// TwinCAT 3 PLC project Test_PLC
// ProgramVersion: 3.1.4026.20
// CompilerDefines: VISU_USEPROPERTYINFO
// libraries:
//   Tc2_Standard, * (Beckhoff Automation GmbH)
//   Tc2_System, * (Beckhoff Automation GmbH)
//   Tc3_Mc3PlanarMotion, * (Beckhoff Automation GmbH)
//   Tc3_Physics, * (Beckhoff Automation GmbH)
//   Tc3_XPlanarUtility, * (Beckhoff Automation GmbH)
//   VisuDialogs, * (System)
// project tree:
//   DUTs/ E_TrackName.TcDUT (not stored), ST_MoverFeedback.TcDUT, U_MoverFeedback.TcDUT
//   / GlobalTextList.TcGTLO, Nc_Task.TcTTO (not stored), PlcTask.TcTTO (not stored), Visualization Manager.TcVMO (not stored)
//   GVLs/ GVL.TcGVL
//   POUs/ FB_StateTrackMove.TcPOU, MAIN.TcPOU
//   VISUs/ TextList_TrackState.TcTLO, Visualization.TcVIS
// real-time tasks:
//   TASK PlcTask: cycle T#10ms, priority 20, ADS port 350
//   TASK Nc Task: cycle T#10ms, priority 1, ADS port 351
//   TASK XPlanar Task_5: cycle T#250us, priority 2, ADS port 352
//   TASK Job Task: cycle default, priority 3
//   TASK MC-Task (MET): cycle T#2ms, priority 4, ADS port 353
//   TASK MC-Task (MPT): cycle T#10ms, priority 5, ADS port 354
//   TASK Job Task_1: cycle default, priority 7
//   TASK MC-Task (MET)_1: cycle T#2ms, priority 8, ADS port 356
//   TASK MC-Task (MPT)_1: cycle T#10ms, priority 9, ADS port 357
//   TASK XPlanar Task_6: cycle T#250us, priority 6, ADS port 355
//   TASK XPlanar Task_7: cycle T#250us, priority 10, ADS port 358
//   TASK EIP Task: cycle T#10ms, priority 12, ADS port 301
// I/O:
//   DEVICE Device 4 (EtherCAT), AmsNetId 169.254.116.218.5.1
//     Term 1 (EK1100) [EK1100 EtherCAT Coupler (2A E-Bus)]
//       Term 2 (EL1008) [EL1008 8Ch. Dig. Input 24V, 3ms]
//       Term 3 (EL2008-0015) [EL2008-0015 8Ch. Dig. Output 24V DC, 0.35A, not short-circuit proof]
//       Term 4 (EL9576) [EL9576 Brake chopper terminal]
//       Term 5 (EL9227-6644) [EL9227-6644 Overcurrent protection 24V DC, 2Ch., 4A/4A, extended functionalities]
//       Term 6 (EL9227-6644) [EL9227-6644 Overcurrent protection 24V DC, 2Ch., 4A/4A, extended functionalities]
//       Term 7 (EL9011) [EL9011 End Terminal]
//   DEVICE Device 5 (EtherCAT), AmsNetId 169.254.116.218.6.1
//     Term 8 (APS4322-7000) [APS4322-7000 Drive]
//       Term 9 (APS4322-5000) [APS4322-5000 Feedback]
//     Term 10 (APS4322-7000) [APS4322-7000 Drive]
//       Term 11 (APS4322-5000) [APS4322-5000 Feedback]
//     Term 12 (APS4322-7000) [APS4322-7000 Drive]
//       Term 13 (APS4322-5000) [APS4322-5000 Feedback]
//     Term 14 (APS4322-7000) [APS4322-7000 Drive]
//       Term 15 (APS4322-5000) [APS4322-5000 Feedback]
//     Term 16 (APS4322-7000) [APS4322-7000 Drive]
//       Term 17 (APS4322-5000) [APS4322-5000 Feedback]
//     Term 18 (APS4322-7000) [APS4322-7000 Drive]
//       Term 19 (APS4322-5000) [APS4322-5000 Feedback]
//   DEVICE Device 6 (RT-Ethernet Adapter)
//   DEVICE Device 1 (TC3 EIP Adapter), AmsNetId 169.254.116.218.2.1
//     Box 20 (TC EtherNet/IP Slave)
// variable links:
//   Device 5 (EtherCAT) <-> TcCOM Objects/XPlanar/Part1/APS4322_P1_1
//     Term 14 (APS4322-7000)/APS Comm Inputs/CommStatusWord <-> Data Pointer/MoverCommStatusWord
//     Term 14 (APS4322-7000)/APS Comm Inputs/Data {1..4} <-> Data Pointer/MoverCommDataIn[{0..3}]  (4 links)
//     Term 14 (APS4322-7000)/APS Comm Outputs/CommControlWord <-> Data Pointer/MoverCommControlWord
//     Term 14 (APS4322-7000)/APS Comm Outputs/Data 1 <-> Data Pointer/MoverCommDataOut
//     Term 14 (APS4322-7000)/APS Diagdata/DC Link Voltage <-> Data Pointer/DcLinkVoltage
//     Term 14 (APS4322-7000)/APS Diagdata/Power supply current <-> Data Pointer/PowerSupplyCurrent
//     Term 14 (APS4322-7000)/APS Inputs/StatusWord <-> Data Pointer/PowerUnitStatusWord
//     Term 14 (APS4322-7000)/APS Outputs/ControlWord <-> Data Pointer/PowerUnitControlWord
//     Term 14 (APS4322-7000)/APS Outputs/Current D 0X0 <-> Data Pointer/DCurrentSetPoints[0]
//     Term 14 (APS4322-7000)/APS Outputs/Current D 0X1 <-> Data Pointer/DCurrentSetPoints[1]
//     Term 14 (APS4322-7000)/APS Outputs/Current D 0X2 <-> Data Pointer/DCurrentSetPoints[2]
//     Term 14 (APS4322-7000)/APS Outputs/Current D 1X0 <-> Data Pointer/DCurrentSetPoints[6]
//     Term 14 (APS4322-7000)/APS Outputs/Current D 1X1 <-> Data Pointer/DCurrentSetPoints[7]
//     Term 14 (APS4322-7000)/APS Outputs/Current D 1X2 <-> Data Pointer/DCurrentSetPoints[8]
//     Term 14 (APS4322-7000)/APS Outputs/Current D 2X0 <-> Data Pointer/DCurrentSetPoints[12]
//     Term 14 (APS4322-7000)/APS Outputs/Current D 2X1 <-> Data Pointer/DCurrentSetPoints[13]
//     Term 14 (APS4322-7000)/APS Outputs/Current D 2X2 <-> Data Pointer/DCurrentSetPoints[14]
//     Term 14 (APS4322-7000)/APS Outputs/Current D 3X0 <-> Data Pointer/DCurrentSetPoints[18]
//     Term 14 (APS4322-7000)/APS Outputs/Current D 3X1 <-> Data Pointer/DCurrentSetPoints[19]
//     Term 14 (APS4322-7000)/APS Outputs/Current D 3X2 <-> Data Pointer/DCurrentSetPoints[20]
//     Term 14 (APS4322-7000)/APS Outputs/Current D 0Y0 <-> Data Pointer/DCurrentSetPoints[3]
//     Term 14 (APS4322-7000)/APS Outputs/Current D 0Y1 <-> Data Pointer/DCurrentSetPoints[4]
//     Term 14 (APS4322-7000)/APS Outputs/Current D 0Y2 <-> Data Pointer/DCurrentSetPoints[5]
//     Term 14 (APS4322-7000)/APS Outputs/Current D 1Y0 <-> Data Pointer/DCurrentSetPoints[9]
//     Term 14 (APS4322-7000)/APS Outputs/Current D 1Y1 <-> Data Pointer/DCurrentSetPoints[10]
//     Term 14 (APS4322-7000)/APS Outputs/Current D 1Y2 <-> Data Pointer/DCurrentSetPoints[11]
//     Term 14 (APS4322-7000)/APS Outputs/Current D 2Y0 <-> Data Pointer/DCurrentSetPoints[15]
//     Term 14 (APS4322-7000)/APS Outputs/Current D 2Y1 <-> Data Pointer/DCurrentSetPoints[16]
//     Term 14 (APS4322-7000)/APS Outputs/Current D 2Y2 <-> Data Pointer/DCurrentSetPoints[17]
//     Term 14 (APS4322-7000)/APS Outputs/Current D 3Y0 <-> Data Pointer/DCurrentSetPoints[21]
//     Term 14 (APS4322-7000)/APS Outputs/Current D 3Y1 <-> Data Pointer/DCurrentSetPoints[22]
//     Term 14 (APS4322-7000)/APS Outputs/Current D 3Y2 <-> Data Pointer/DCurrentSetPoints[23]
//     Term 14 (APS4322-7000)/APS Outputs/Current Q 0X0 <-> Data Pointer/QCurrentSetPoints[0]
//     Term 14 (APS4322-7000)/APS Outputs/Current Q 0X1 <-> Data Pointer/QCurrentSetPoints[1]
//     Term 14 (APS4322-7000)/APS Outputs/Current Q 0X2 <-> Data Pointer/QCurrentSetPoints[2]
//     Term 14 (APS4322-7000)/APS Outputs/Current Q 1X0 <-> Data Pointer/QCurrentSetPoints[6]
//     Term 14 (APS4322-7000)/APS Outputs/Current Q 1X1 <-> Data Pointer/QCurrentSetPoints[7]
//     Term 14 (APS4322-7000)/APS Outputs/Current Q 1X2 <-> Data Pointer/QCurrentSetPoints[8]
//     Term 14 (APS4322-7000)/APS Outputs/Current Q 2X0 <-> Data Pointer/QCurrentSetPoints[12]
//     Term 14 (APS4322-7000)/APS Outputs/Current Q 2X1 <-> Data Pointer/QCurrentSetPoints[13]
//     Term 14 (APS4322-7000)/APS Outputs/Current Q 2X2 <-> Data Pointer/QCurrentSetPoints[14]
//     Term 14 (APS4322-7000)/APS Outputs/Current Q 3X0 <-> Data Pointer/QCurrentSetPoints[18]
//     Term 14 (APS4322-7000)/APS Outputs/Current Q 3X1 <-> Data Pointer/QCurrentSetPoints[19]
//     Term 14 (APS4322-7000)/APS Outputs/Current Q 3X2 <-> Data Pointer/QCurrentSetPoints[20]
//     Term 14 (APS4322-7000)/APS Outputs/Current Q 0Y0 <-> Data Pointer/QCurrentSetPoints[3]
//     Term 14 (APS4322-7000)/APS Outputs/Current Q 0Y1 <-> Data Pointer/QCurrentSetPoints[4]
//     Term 14 (APS4322-7000)/APS Outputs/Current Q 0Y2 <-> Data Pointer/QCurrentSetPoints[5]
//     Term 14 (APS4322-7000)/APS Outputs/Current Q 1Y0 <-> Data Pointer/QCurrentSetPoints[9]
//     Term 14 (APS4322-7000)/APS Outputs/Current Q 1Y1 <-> Data Pointer/QCurrentSetPoints[10]
//     Term 14 (APS4322-7000)/APS Outputs/Current Q 1Y2 <-> Data Pointer/QCurrentSetPoints[11]
//     Term 14 (APS4322-7000)/APS Outputs/Current Q 2Y0 <-> Data Pointer/QCurrentSetPoints[15]
//     Term 14 (APS4322-7000)/APS Outputs/Current Q 2Y1 <-> Data Pointer/QCurrentSetPoints[16]
//     Term 14 (APS4322-7000)/APS Outputs/Current Q 2Y2 <-> Data Pointer/QCurrentSetPoints[17]
//     Term 14 (APS4322-7000)/APS Outputs/Current Q 3Y0 <-> Data Pointer/QCurrentSetPoints[21]
//     Term 14 (APS4322-7000)/APS Outputs/Current Q 3Y1 <-> Data Pointer/QCurrentSetPoints[22]
//     Term 14 (APS4322-7000)/APS Outputs/Current Q 3Y2 <-> Data Pointer/QCurrentSetPoints[23]
//     Term 14 (APS4322-7000)/APS Outputs/PhiE 0X0 <-> Data Pointer/PhiSetPoints[0]
//     Term 14 (APS4322-7000)/APS Outputs/PhiE 0X1 <-> Data Pointer/PhiSetPoints[1]
//     Term 14 (APS4322-7000)/APS Outputs/PhiE 0X2 <-> Data Pointer/PhiSetPoints[2]
//     Term 14 (APS4322-7000)/APS Outputs/PhiE 1X0 <-> Data Pointer/PhiSetPoints[6]
//     Term 14 (APS4322-7000)/APS Outputs/PhiE 1X1 <-> Data Pointer/PhiSetPoints[7]
//     Term 14 (APS4322-7000)/APS Outputs/PhiE 1X2 <-> Data Pointer/PhiSetPoints[8]
//     Term 14 (APS4322-7000)/APS Outputs/PhiE 2X0 <-> Data Pointer/PhiSetPoints[12]
//     Term 14 (APS4322-7000)/APS Outputs/PhiE 2X1 <-> Data Pointer/PhiSetPoints[13]
//     Term 14 (APS4322-7000)/APS Outputs/PhiE 2X2 <-> Data Pointer/PhiSetPoints[14]
//     Term 14 (APS4322-7000)/APS Outputs/PhiE 3X0 <-> Data Pointer/PhiSetPoints[18]
//     Term 14 (APS4322-7000)/APS Outputs/PhiE 3X1 <-> Data Pointer/PhiSetPoints[19]
//     Term 14 (APS4322-7000)/APS Outputs/PhiE 3X2 <-> Data Pointer/PhiSetPoints[20]
//     Term 14 (APS4322-7000)/APS Outputs/PhiE 0Y0 <-> Data Pointer/PhiSetPoints[3]
//     Term 14 (APS4322-7000)/APS Outputs/PhiE 0Y1 <-> Data Pointer/PhiSetPoints[4]
//     Term 14 (APS4322-7000)/APS Outputs/PhiE 0Y2 <-> Data Pointer/PhiSetPoints[5]
//     Term 14 (APS4322-7000)/APS Outputs/PhiE 1Y0 <-> Data Pointer/PhiSetPoints[9]
//     Term 14 (APS4322-7000)/APS Outputs/PhiE 1Y1 <-> Data Pointer/PhiSetPoints[10]
//     Term 14 (APS4322-7000)/APS Outputs/PhiE 1Y2 <-> Data Pointer/PhiSetPoints[11]
//     Term 14 (APS4322-7000)/APS Outputs/PhiE 2Y0 <-> Data Pointer/PhiSetPoints[15]
//     Term 14 (APS4322-7000)/APS Outputs/PhiE 2Y1 <-> Data Pointer/PhiSetPoints[16]
//     Term 14 (APS4322-7000)/APS Outputs/PhiE 2Y2 <-> Data Pointer/PhiSetPoints[17]
//     Term 14 (APS4322-7000)/APS Outputs/PhiE 3Y0 <-> Data Pointer/PhiSetPoints[21]
//     Term 14 (APS4322-7000)/APS Outputs/PhiE 3Y1 <-> Data Pointer/PhiSetPoints[22]
//     Term 14 (APS4322-7000)/APS Outputs/PhiE 3Y2 <-> Data Pointer/PhiSetPoints[23]
//     Term 14 (APS4322-7000)/Term 15 (APS4322-5000)/FB Inputs/A{0..8 step 2} X-Field <-> Data Pointer/HallSensorFieldsXYZ[{0..12 step 3}]  (5 links)
//     Term 14 (APS4322-7000)/Term 15 (APS4322-5000)/FB Inputs/A{0..8 step 2} Y-Field <-> Data Pointer/HallSensorFieldsXYZ[{1..13 step 3}]  (5 links)
//     Term 14 (APS4322-7000)/Term 15 (APS4322-5000)/FB Inputs/A{0..8 step 2} Z-Field <-> Data Pointer/HallSensorFieldsXYZ[{2..14 step 3}]  (5 links)
//     Term 14 (APS4322-7000)/Term 15 (APS4322-5000)/FB Inputs/B{1..9 step 2} X-Field <-> Data Pointer/HallSensorFieldsXYZ[{15..27 step 3}]  (5 links)
//     Term 14 (APS4322-7000)/Term 15 (APS4322-5000)/FB Inputs/B{1..9 step 2} Y-Field <-> Data Pointer/HallSensorFieldsXYZ[{16..28 step 3}]  (5 links)
//     Term 14 (APS4322-7000)/Term 15 (APS4322-5000)/FB Inputs/B{1..9 step 2} Z-Field <-> Data Pointer/HallSensorFieldsXYZ[{17..29 step 3}]  (5 links)
//     Term 14 (APS4322-7000)/Term 15 (APS4322-5000)/FB Inputs/C{0..8 step 2} X-Field <-> Data Pointer/HallSensorFieldsXYZ[{30..42 step 3}]  (5 links)
//     Term 14 (APS4322-7000)/Term 15 (APS4322-5000)/FB Inputs/C{0..8 step 2} Y-Field <-> Data Pointer/HallSensorFieldsXYZ[{31..43 step 3}]  (5 links)
//     Term 14 (APS4322-7000)/Term 15 (APS4322-5000)/FB Inputs/C{0..8 step 2} Z-Field <-> Data Pointer/HallSensorFieldsXYZ[{32..44 step 3}]  (5 links)
//     Term 14 (APS4322-7000)/Term 15 (APS4322-5000)/FB Inputs/D{1..9 step 2} X-Field <-> Data Pointer/HallSensorFieldsXYZ[{45..57 step 3}]  (5 links)
//     Term 14 (APS4322-7000)/Term 15 (APS4322-5000)/FB Inputs/D{1..9 step 2} Y-Field <-> Data Pointer/HallSensorFieldsXYZ[{46..58 step 3}]  (5 links)
//     Term 14 (APS4322-7000)/Term 15 (APS4322-5000)/FB Inputs/D{1..9 step 2} Z-Field <-> Data Pointer/HallSensorFieldsXYZ[{47..59 step 3}]  (5 links)
//     Term 14 (APS4322-7000)/Term 15 (APS4322-5000)/FB Inputs/E{0..8 step 2} X-Field <-> Data Pointer/HallSensorFieldsXYZ[{60..72 step 3}]  (5 links)
//     Term 14 (APS4322-7000)/Term 15 (APS4322-5000)/FB Inputs/E{0..8 step 2} Y-Field <-> Data Pointer/HallSensorFieldsXYZ[{61..73 step 3}]  (5 links)
//     Term 14 (APS4322-7000)/Term 15 (APS4322-5000)/FB Inputs/E{0..8 step 2} Z-Field <-> Data Pointer/HallSensorFieldsXYZ[{62..74 step 3}]  (5 links)
//     Term 14 (APS4322-7000)/Term 15 (APS4322-5000)/FB Inputs/F{1..9 step 2} X-Field <-> Data Pointer/HallSensorFieldsXYZ[{75..87 step 3}]  (5 links)
//     Term 14 (APS4322-7000)/Term 15 (APS4322-5000)/FB Inputs/F{1..9 step 2} Y-Field <-> Data Pointer/HallSensorFieldsXYZ[{76..88 step 3}]  (5 links)
//     Term 14 (APS4322-7000)/Term 15 (APS4322-5000)/FB Inputs/F{1..9 step 2} Z-Field <-> Data Pointer/HallSensorFieldsXYZ[{77..89 step 3}]  (5 links)
//     Term 14 (APS4322-7000)/Term 15 (APS4322-5000)/FB Inputs/G{0..8 step 2} X-Field <-> Data Pointer/HallSensorFieldsXYZ[{90..102 step 3}]  (5 links)
//     Term 14 (APS4322-7000)/Term 15 (APS4322-5000)/FB Inputs/G{0..8 step 2} Y-Field <-> Data Pointer/HallSensorFieldsXYZ[{91..103 step 3}]  (5 links)
//     Term 14 (APS4322-7000)/Term 15 (APS4322-5000)/FB Inputs/G{0..8 step 2} Z-Field <-> Data Pointer/HallSensorFieldsXYZ[{92..104 step 3}]  (5 links)
//     Term 14 (APS4322-7000)/Term 15 (APS4322-5000)/FB Inputs/H{1..9 step 2} X-Field <-> Data Pointer/HallSensorFieldsXYZ[{105..117 step 3}]  (5 links)
//     Term 14 (APS4322-7000)/Term 15 (APS4322-5000)/FB Inputs/H{1..9 step 2} Y-Field <-> Data Pointer/HallSensorFieldsXYZ[{106..118 step 3}]  (5 links)
//     Term 14 (APS4322-7000)/Term 15 (APS4322-5000)/FB Inputs/H{1..9 step 2} Z-Field <-> Data Pointer/HallSensorFieldsXYZ[{107..119 step 3}]  (5 links)
//     Term 14 (APS4322-7000)/Term 15 (APS4322-5000)/FB Inputs/I{0..8 step 2} X-Field <-> Data Pointer/HallSensorFieldsXYZ[{120..132 step 3}]  (5 links)
//     Term 14 (APS4322-7000)/Term 15 (APS4322-5000)/FB Inputs/I{0..8 step 2} Y-Field <-> Data Pointer/HallSensorFieldsXYZ[{121..133 step 3}]  (5 links)
//     Term 14 (APS4322-7000)/Term 15 (APS4322-5000)/FB Inputs/I{0..8 step 2} Z-Field <-> Data Pointer/HallSensorFieldsXYZ[{122..134 step 3}]  (5 links)
//     Term 14 (APS4322-7000)/Term 15 (APS4322-5000)/FB Inputs/J{1..9 step 2} X-Field <-> Data Pointer/HallSensorFieldsXYZ[{135..147 step 3}]  (5 links)
//     Term 14 (APS4322-7000)/Term 15 (APS4322-5000)/FB Inputs/J{1..9 step 2} Y-Field <-> Data Pointer/HallSensorFieldsXYZ[{136..148 step 3}]  (5 links)
//     Term 14 (APS4322-7000)/Term 15 (APS4322-5000)/FB Inputs/J{1..9 step 2} Z-Field <-> Data Pointer/HallSensorFieldsXYZ[{137..149 step 3}]  (5 links)
//     Term 14 (APS4322-7000)/Term 15 (APS4322-5000)/FB Inputs/Status <-> Data Pointer/FeedbackStatus
//   Device 5 (EtherCAT) <-> TcCOM Objects/XPlanar/Part1/APS4322_P1_2
//     Term 16 (APS4322-7000)/APS Comm Inputs/CommStatusWord <-> Data Pointer/MoverCommStatusWord
//     Term 16 (APS4322-7000)/APS Comm Inputs/Data {1..4} <-> Data Pointer/MoverCommDataIn[{0..3}]  (4 links)
//     Term 16 (APS4322-7000)/APS Comm Outputs/CommControlWord <-> Data Pointer/MoverCommControlWord
//     Term 16 (APS4322-7000)/APS Comm Outputs/Data 1 <-> Data Pointer/MoverCommDataOut
//     Term 16 (APS4322-7000)/APS Diagdata/DC Link Voltage <-> Data Pointer/DcLinkVoltage
//     Term 16 (APS4322-7000)/APS Diagdata/Power supply current <-> Data Pointer/PowerSupplyCurrent
//     Term 16 (APS4322-7000)/APS Inputs/StatusWord <-> Data Pointer/PowerUnitStatusWord
//     Term 16 (APS4322-7000)/APS Outputs/ControlWord <-> Data Pointer/PowerUnitControlWord
//     Term 16 (APS4322-7000)/APS Outputs/Current D 0X0 <-> Data Pointer/DCurrentSetPoints[0]
//     Term 16 (APS4322-7000)/APS Outputs/Current D 0X1 <-> Data Pointer/DCurrentSetPoints[1]
//     Term 16 (APS4322-7000)/APS Outputs/Current D 0X2 <-> Data Pointer/DCurrentSetPoints[2]
//     Term 16 (APS4322-7000)/APS Outputs/Current D 1X0 <-> Data Pointer/DCurrentSetPoints[6]
//     Term 16 (APS4322-7000)/APS Outputs/Current D 1X1 <-> Data Pointer/DCurrentSetPoints[7]
//     Term 16 (APS4322-7000)/APS Outputs/Current D 1X2 <-> Data Pointer/DCurrentSetPoints[8]
//     Term 16 (APS4322-7000)/APS Outputs/Current D 2X0 <-> Data Pointer/DCurrentSetPoints[12]
//     Term 16 (APS4322-7000)/APS Outputs/Current D 2X1 <-> Data Pointer/DCurrentSetPoints[13]
//     Term 16 (APS4322-7000)/APS Outputs/Current D 2X2 <-> Data Pointer/DCurrentSetPoints[14]
//     Term 16 (APS4322-7000)/APS Outputs/Current D 3X0 <-> Data Pointer/DCurrentSetPoints[18]
//     Term 16 (APS4322-7000)/APS Outputs/Current D 3X1 <-> Data Pointer/DCurrentSetPoints[19]
//     Term 16 (APS4322-7000)/APS Outputs/Current D 3X2 <-> Data Pointer/DCurrentSetPoints[20]
//     Term 16 (APS4322-7000)/APS Outputs/Current D 0Y0 <-> Data Pointer/DCurrentSetPoints[3]
//     Term 16 (APS4322-7000)/APS Outputs/Current D 0Y1 <-> Data Pointer/DCurrentSetPoints[4]
//     Term 16 (APS4322-7000)/APS Outputs/Current D 0Y2 <-> Data Pointer/DCurrentSetPoints[5]
//     Term 16 (APS4322-7000)/APS Outputs/Current D 1Y0 <-> Data Pointer/DCurrentSetPoints[9]
//     Term 16 (APS4322-7000)/APS Outputs/Current D 1Y1 <-> Data Pointer/DCurrentSetPoints[10]
//     Term 16 (APS4322-7000)/APS Outputs/Current D 1Y2 <-> Data Pointer/DCurrentSetPoints[11]
//     Term 16 (APS4322-7000)/APS Outputs/Current D 2Y0 <-> Data Pointer/DCurrentSetPoints[15]
//     Term 16 (APS4322-7000)/APS Outputs/Current D 2Y1 <-> Data Pointer/DCurrentSetPoints[16]
//     Term 16 (APS4322-7000)/APS Outputs/Current D 2Y2 <-> Data Pointer/DCurrentSetPoints[17]
//     Term 16 (APS4322-7000)/APS Outputs/Current D 3Y0 <-> Data Pointer/DCurrentSetPoints[21]
//     Term 16 (APS4322-7000)/APS Outputs/Current D 3Y1 <-> Data Pointer/DCurrentSetPoints[22]
//     Term 16 (APS4322-7000)/APS Outputs/Current D 3Y2 <-> Data Pointer/DCurrentSetPoints[23]
//     Term 16 (APS4322-7000)/APS Outputs/Current Q 0X0 <-> Data Pointer/QCurrentSetPoints[0]
//     Term 16 (APS4322-7000)/APS Outputs/Current Q 0X1 <-> Data Pointer/QCurrentSetPoints[1]
//     Term 16 (APS4322-7000)/APS Outputs/Current Q 0X2 <-> Data Pointer/QCurrentSetPoints[2]
//     Term 16 (APS4322-7000)/APS Outputs/Current Q 1X0 <-> Data Pointer/QCurrentSetPoints[6]
//     Term 16 (APS4322-7000)/APS Outputs/Current Q 1X1 <-> Data Pointer/QCurrentSetPoints[7]
//     Term 16 (APS4322-7000)/APS Outputs/Current Q 1X2 <-> Data Pointer/QCurrentSetPoints[8]
//     Term 16 (APS4322-7000)/APS Outputs/Current Q 2X0 <-> Data Pointer/QCurrentSetPoints[12]
//     Term 16 (APS4322-7000)/APS Outputs/Current Q 2X1 <-> Data Pointer/QCurrentSetPoints[13]
//     Term 16 (APS4322-7000)/APS Outputs/Current Q 2X2 <-> Data Pointer/QCurrentSetPoints[14]
//     Term 16 (APS4322-7000)/APS Outputs/Current Q 3X0 <-> Data Pointer/QCurrentSetPoints[18]
//     Term 16 (APS4322-7000)/APS Outputs/Current Q 3X1 <-> Data Pointer/QCurrentSetPoints[19]
//     Term 16 (APS4322-7000)/APS Outputs/Current Q 3X2 <-> Data Pointer/QCurrentSetPoints[20]
//     Term 16 (APS4322-7000)/APS Outputs/Current Q 0Y0 <-> Data Pointer/QCurrentSetPoints[3]
//     Term 16 (APS4322-7000)/APS Outputs/Current Q 0Y1 <-> Data Pointer/QCurrentSetPoints[4]
//     Term 16 (APS4322-7000)/APS Outputs/Current Q 0Y2 <-> Data Pointer/QCurrentSetPoints[5]
//     Term 16 (APS4322-7000)/APS Outputs/Current Q 1Y0 <-> Data Pointer/QCurrentSetPoints[9]
//     Term 16 (APS4322-7000)/APS Outputs/Current Q 1Y1 <-> Data Pointer/QCurrentSetPoints[10]
//     Term 16 (APS4322-7000)/APS Outputs/Current Q 1Y2 <-> Data Pointer/QCurrentSetPoints[11]
//     Term 16 (APS4322-7000)/APS Outputs/Current Q 2Y0 <-> Data Pointer/QCurrentSetPoints[15]
//     Term 16 (APS4322-7000)/APS Outputs/Current Q 2Y1 <-> Data Pointer/QCurrentSetPoints[16]
//     Term 16 (APS4322-7000)/APS Outputs/Current Q 2Y2 <-> Data Pointer/QCurrentSetPoints[17]
//     Term 16 (APS4322-7000)/APS Outputs/Current Q 3Y0 <-> Data Pointer/QCurrentSetPoints[21]
//     Term 16 (APS4322-7000)/APS Outputs/Current Q 3Y1 <-> Data Pointer/QCurrentSetPoints[22]
//     Term 16 (APS4322-7000)/APS Outputs/Current Q 3Y2 <-> Data Pointer/QCurrentSetPoints[23]
//     Term 16 (APS4322-7000)/APS Outputs/PhiE 0X0 <-> Data Pointer/PhiSetPoints[0]
//     Term 16 (APS4322-7000)/APS Outputs/PhiE 0X1 <-> Data Pointer/PhiSetPoints[1]
//     Term 16 (APS4322-7000)/APS Outputs/PhiE 0X2 <-> Data Pointer/PhiSetPoints[2]
//     Term 16 (APS4322-7000)/APS Outputs/PhiE 1X0 <-> Data Pointer/PhiSetPoints[6]
//     Term 16 (APS4322-7000)/APS Outputs/PhiE 1X1 <-> Data Pointer/PhiSetPoints[7]
//     Term 16 (APS4322-7000)/APS Outputs/PhiE 1X2 <-> Data Pointer/PhiSetPoints[8]
//     Term 16 (APS4322-7000)/APS Outputs/PhiE 2X0 <-> Data Pointer/PhiSetPoints[12]
//     Term 16 (APS4322-7000)/APS Outputs/PhiE 2X1 <-> Data Pointer/PhiSetPoints[13]
//     Term 16 (APS4322-7000)/APS Outputs/PhiE 2X2 <-> Data Pointer/PhiSetPoints[14]
//     Term 16 (APS4322-7000)/APS Outputs/PhiE 3X0 <-> Data Pointer/PhiSetPoints[18]
//     Term 16 (APS4322-7000)/APS Outputs/PhiE 3X1 <-> Data Pointer/PhiSetPoints[19]
//     Term 16 (APS4322-7000)/APS Outputs/PhiE 3X2 <-> Data Pointer/PhiSetPoints[20]
//     Term 16 (APS4322-7000)/APS Outputs/PhiE 0Y0 <-> Data Pointer/PhiSetPoints[3]
//     Term 16 (APS4322-7000)/APS Outputs/PhiE 0Y1 <-> Data Pointer/PhiSetPoints[4]
//     Term 16 (APS4322-7000)/APS Outputs/PhiE 0Y2 <-> Data Pointer/PhiSetPoints[5]
//     Term 16 (APS4322-7000)/APS Outputs/PhiE 1Y0 <-> Data Pointer/PhiSetPoints[9]
//     Term 16 (APS4322-7000)/APS Outputs/PhiE 1Y1 <-> Data Pointer/PhiSetPoints[10]
//     Term 16 (APS4322-7000)/APS Outputs/PhiE 1Y2 <-> Data Pointer/PhiSetPoints[11]
//     Term 16 (APS4322-7000)/APS Outputs/PhiE 2Y0 <-> Data Pointer/PhiSetPoints[15]
//     Term 16 (APS4322-7000)/APS Outputs/PhiE 2Y1 <-> Data Pointer/PhiSetPoints[16]
//     Term 16 (APS4322-7000)/APS Outputs/PhiE 2Y2 <-> Data Pointer/PhiSetPoints[17]
//     Term 16 (APS4322-7000)/APS Outputs/PhiE 3Y0 <-> Data Pointer/PhiSetPoints[21]
//     Term 16 (APS4322-7000)/APS Outputs/PhiE 3Y1 <-> Data Pointer/PhiSetPoints[22]
//     Term 16 (APS4322-7000)/APS Outputs/PhiE 3Y2 <-> Data Pointer/PhiSetPoints[23]
//     Term 16 (APS4322-7000)/Term 17 (APS4322-5000)/FB Inputs/A{0..8 step 2} X-Field <-> Data Pointer/HallSensorFieldsXYZ[{0..12 step 3}]  (5 links)
//     Term 16 (APS4322-7000)/Term 17 (APS4322-5000)/FB Inputs/A{0..8 step 2} Y-Field <-> Data Pointer/HallSensorFieldsXYZ[{1..13 step 3}]  (5 links)
//     Term 16 (APS4322-7000)/Term 17 (APS4322-5000)/FB Inputs/A{0..8 step 2} Z-Field <-> Data Pointer/HallSensorFieldsXYZ[{2..14 step 3}]  (5 links)
//     Term 16 (APS4322-7000)/Term 17 (APS4322-5000)/FB Inputs/B{1..9 step 2} X-Field <-> Data Pointer/HallSensorFieldsXYZ[{15..27 step 3}]  (5 links)
//     Term 16 (APS4322-7000)/Term 17 (APS4322-5000)/FB Inputs/B{1..9 step 2} Y-Field <-> Data Pointer/HallSensorFieldsXYZ[{16..28 step 3}]  (5 links)
//     Term 16 (APS4322-7000)/Term 17 (APS4322-5000)/FB Inputs/B{1..9 step 2} Z-Field <-> Data Pointer/HallSensorFieldsXYZ[{17..29 step 3}]  (5 links)
//     Term 16 (APS4322-7000)/Term 17 (APS4322-5000)/FB Inputs/C{0..8 step 2} X-Field <-> Data Pointer/HallSensorFieldsXYZ[{30..42 step 3}]  (5 links)
//     Term 16 (APS4322-7000)/Term 17 (APS4322-5000)/FB Inputs/C{0..8 step 2} Y-Field <-> Data Pointer/HallSensorFieldsXYZ[{31..43 step 3}]  (5 links)
//     Term 16 (APS4322-7000)/Term 17 (APS4322-5000)/FB Inputs/C{0..8 step 2} Z-Field <-> Data Pointer/HallSensorFieldsXYZ[{32..44 step 3}]  (5 links)
//     Term 16 (APS4322-7000)/Term 17 (APS4322-5000)/FB Inputs/D{1..9 step 2} X-Field <-> Data Pointer/HallSensorFieldsXYZ[{45..57 step 3}]  (5 links)
//     Term 16 (APS4322-7000)/Term 17 (APS4322-5000)/FB Inputs/D{1..9 step 2} Y-Field <-> Data Pointer/HallSensorFieldsXYZ[{46..58 step 3}]  (5 links)
//     Term 16 (APS4322-7000)/Term 17 (APS4322-5000)/FB Inputs/D{1..9 step 2} Z-Field <-> Data Pointer/HallSensorFieldsXYZ[{47..59 step 3}]  (5 links)
//     Term 16 (APS4322-7000)/Term 17 (APS4322-5000)/FB Inputs/E{0..8 step 2} X-Field <-> Data Pointer/HallSensorFieldsXYZ[{60..72 step 3}]  (5 links)
//     Term 16 (APS4322-7000)/Term 17 (APS4322-5000)/FB Inputs/E{0..8 step 2} Y-Field <-> Data Pointer/HallSensorFieldsXYZ[{61..73 step 3}]  (5 links)
//     Term 16 (APS4322-7000)/Term 17 (APS4322-5000)/FB Inputs/E{0..8 step 2} Z-Field <-> Data Pointer/HallSensorFieldsXYZ[{62..74 step 3}]  (5 links)
//     Term 16 (APS4322-7000)/Term 17 (APS4322-5000)/FB Inputs/F{1..9 step 2} X-Field <-> Data Pointer/HallSensorFieldsXYZ[{75..87 step 3}]  (5 links)
//     Term 16 (APS4322-7000)/Term 17 (APS4322-5000)/FB Inputs/F{1..9 step 2} Y-Field <-> Data Pointer/HallSensorFieldsXYZ[{76..88 step 3}]  (5 links)
//     Term 16 (APS4322-7000)/Term 17 (APS4322-5000)/FB Inputs/F{1..9 step 2} Z-Field <-> Data Pointer/HallSensorFieldsXYZ[{77..89 step 3}]  (5 links)
//     Term 16 (APS4322-7000)/Term 17 (APS4322-5000)/FB Inputs/G{0..8 step 2} X-Field <-> Data Pointer/HallSensorFieldsXYZ[{90..102 step 3}]  (5 links)
//     Term 16 (APS4322-7000)/Term 17 (APS4322-5000)/FB Inputs/G{0..8 step 2} Y-Field <-> Data Pointer/HallSensorFieldsXYZ[{91..103 step 3}]  (5 links)
//     Term 16 (APS4322-7000)/Term 17 (APS4322-5000)/FB Inputs/G{0..8 step 2} Z-Field <-> Data Pointer/HallSensorFieldsXYZ[{92..104 step 3}]  (5 links)
//     Term 16 (APS4322-7000)/Term 17 (APS4322-5000)/FB Inputs/H{1..9 step 2} X-Field <-> Data Pointer/HallSensorFieldsXYZ[{105..117 step 3}]  (5 links)
//     Term 16 (APS4322-7000)/Term 17 (APS4322-5000)/FB Inputs/H{1..9 step 2} Y-Field <-> Data Pointer/HallSensorFieldsXYZ[{106..118 step 3}]  (5 links)
//     Term 16 (APS4322-7000)/Term 17 (APS4322-5000)/FB Inputs/H{1..9 step 2} Z-Field <-> Data Pointer/HallSensorFieldsXYZ[{107..119 step 3}]  (5 links)
//     Term 16 (APS4322-7000)/Term 17 (APS4322-5000)/FB Inputs/I{0..8 step 2} X-Field <-> Data Pointer/HallSensorFieldsXYZ[{120..132 step 3}]  (5 links)
//     Term 16 (APS4322-7000)/Term 17 (APS4322-5000)/FB Inputs/I{0..8 step 2} Y-Field <-> Data Pointer/HallSensorFieldsXYZ[{121..133 step 3}]  (5 links)
//     Term 16 (APS4322-7000)/Term 17 (APS4322-5000)/FB Inputs/I{0..8 step 2} Z-Field <-> Data Pointer/HallSensorFieldsXYZ[{122..134 step 3}]  (5 links)
//     Term 16 (APS4322-7000)/Term 17 (APS4322-5000)/FB Inputs/J{1..9 step 2} X-Field <-> Data Pointer/HallSensorFieldsXYZ[{135..147 step 3}]  (5 links)
//     Term 16 (APS4322-7000)/Term 17 (APS4322-5000)/FB Inputs/J{1..9 step 2} Y-Field <-> Data Pointer/HallSensorFieldsXYZ[{136..148 step 3}]  (5 links)
//     Term 16 (APS4322-7000)/Term 17 (APS4322-5000)/FB Inputs/J{1..9 step 2} Z-Field <-> Data Pointer/HallSensorFieldsXYZ[{137..149 step 3}]  (5 links)
//     Term 16 (APS4322-7000)/Term 17 (APS4322-5000)/FB Inputs/Status <-> Data Pointer/FeedbackStatus
//   Device 5 (EtherCAT) <-> TcCOM Objects/XPlanar/Part1/APS4322_P1_3
//     Term 18 (APS4322-7000)/APS Comm Inputs/CommStatusWord <-> Data Pointer/MoverCommStatusWord
//     Term 18 (APS4322-7000)/APS Comm Inputs/Data {1..4} <-> Data Pointer/MoverCommDataIn[{0..3}]  (4 links)
//     Term 18 (APS4322-7000)/APS Comm Outputs/CommControlWord <-> Data Pointer/MoverCommControlWord
//     Term 18 (APS4322-7000)/APS Comm Outputs/Data 1 <-> Data Pointer/MoverCommDataOut
//     Term 18 (APS4322-7000)/APS Diagdata/DC Link Voltage <-> Data Pointer/DcLinkVoltage
//     Term 18 (APS4322-7000)/APS Diagdata/Power supply current <-> Data Pointer/PowerSupplyCurrent
//     Term 18 (APS4322-7000)/APS Inputs/StatusWord <-> Data Pointer/PowerUnitStatusWord
//     Term 18 (APS4322-7000)/APS Outputs/ControlWord <-> Data Pointer/PowerUnitControlWord
//     Term 18 (APS4322-7000)/APS Outputs/Current D 0X0 <-> Data Pointer/DCurrentSetPoints[0]
//     Term 18 (APS4322-7000)/APS Outputs/Current D 0X1 <-> Data Pointer/DCurrentSetPoints[1]
//     Term 18 (APS4322-7000)/APS Outputs/Current D 0X2 <-> Data Pointer/DCurrentSetPoints[2]
//     Term 18 (APS4322-7000)/APS Outputs/Current D 1X0 <-> Data Pointer/DCurrentSetPoints[6]
//     Term 18 (APS4322-7000)/APS Outputs/Current D 1X1 <-> Data Pointer/DCurrentSetPoints[7]
//     Term 18 (APS4322-7000)/APS Outputs/Current D 1X2 <-> Data Pointer/DCurrentSetPoints[8]
//     Term 18 (APS4322-7000)/APS Outputs/Current D 2X0 <-> Data Pointer/DCurrentSetPoints[12]
//     Term 18 (APS4322-7000)/APS Outputs/Current D 2X1 <-> Data Pointer/DCurrentSetPoints[13]
//     Term 18 (APS4322-7000)/APS Outputs/Current D 2X2 <-> Data Pointer/DCurrentSetPoints[14]
//     Term 18 (APS4322-7000)/APS Outputs/Current D 3X0 <-> Data Pointer/DCurrentSetPoints[18]
//     Term 18 (APS4322-7000)/APS Outputs/Current D 3X1 <-> Data Pointer/DCurrentSetPoints[19]
//     Term 18 (APS4322-7000)/APS Outputs/Current D 3X2 <-> Data Pointer/DCurrentSetPoints[20]
//     Term 18 (APS4322-7000)/APS Outputs/Current D 0Y0 <-> Data Pointer/DCurrentSetPoints[3]
//     Term 18 (APS4322-7000)/APS Outputs/Current D 0Y1 <-> Data Pointer/DCurrentSetPoints[4]
//     Term 18 (APS4322-7000)/APS Outputs/Current D 0Y2 <-> Data Pointer/DCurrentSetPoints[5]
//     Term 18 (APS4322-7000)/APS Outputs/Current D 1Y0 <-> Data Pointer/DCurrentSetPoints[9]
//     Term 18 (APS4322-7000)/APS Outputs/Current D 1Y1 <-> Data Pointer/DCurrentSetPoints[10]
//     Term 18 (APS4322-7000)/APS Outputs/Current D 1Y2 <-> Data Pointer/DCurrentSetPoints[11]
//     Term 18 (APS4322-7000)/APS Outputs/Current D 2Y0 <-> Data Pointer/DCurrentSetPoints[15]
//     Term 18 (APS4322-7000)/APS Outputs/Current D 2Y1 <-> Data Pointer/DCurrentSetPoints[16]
//     Term 18 (APS4322-7000)/APS Outputs/Current D 2Y2 <-> Data Pointer/DCurrentSetPoints[17]
//     Term 18 (APS4322-7000)/APS Outputs/Current D 3Y0 <-> Data Pointer/DCurrentSetPoints[21]
//     Term 18 (APS4322-7000)/APS Outputs/Current D 3Y1 <-> Data Pointer/DCurrentSetPoints[22]
//     Term 18 (APS4322-7000)/APS Outputs/Current D 3Y2 <-> Data Pointer/DCurrentSetPoints[23]
//     Term 18 (APS4322-7000)/APS Outputs/Current Q 0X0 <-> Data Pointer/QCurrentSetPoints[0]
//     Term 18 (APS4322-7000)/APS Outputs/Current Q 0X1 <-> Data Pointer/QCurrentSetPoints[1]
//     Term 18 (APS4322-7000)/APS Outputs/Current Q 0X2 <-> Data Pointer/QCurrentSetPoints[2]
//     Term 18 (APS4322-7000)/APS Outputs/Current Q 1X0 <-> Data Pointer/QCurrentSetPoints[6]
//     Term 18 (APS4322-7000)/APS Outputs/Current Q 1X1 <-> Data Pointer/QCurrentSetPoints[7]
//     Term 18 (APS4322-7000)/APS Outputs/Current Q 1X2 <-> Data Pointer/QCurrentSetPoints[8]
//     Term 18 (APS4322-7000)/APS Outputs/Current Q 2X0 <-> Data Pointer/QCurrentSetPoints[12]
//     Term 18 (APS4322-7000)/APS Outputs/Current Q 2X1 <-> Data Pointer/QCurrentSetPoints[13]
//     Term 18 (APS4322-7000)/APS Outputs/Current Q 2X2 <-> Data Pointer/QCurrentSetPoints[14]
//     Term 18 (APS4322-7000)/APS Outputs/Current Q 3X0 <-> Data Pointer/QCurrentSetPoints[18]
//     Term 18 (APS4322-7000)/APS Outputs/Current Q 3X1 <-> Data Pointer/QCurrentSetPoints[19]
//     Term 18 (APS4322-7000)/APS Outputs/Current Q 3X2 <-> Data Pointer/QCurrentSetPoints[20]
//     Term 18 (APS4322-7000)/APS Outputs/Current Q 0Y0 <-> Data Pointer/QCurrentSetPoints[3]
//     Term 18 (APS4322-7000)/APS Outputs/Current Q 0Y1 <-> Data Pointer/QCurrentSetPoints[4]
//     Term 18 (APS4322-7000)/APS Outputs/Current Q 0Y2 <-> Data Pointer/QCurrentSetPoints[5]
//     Term 18 (APS4322-7000)/APS Outputs/Current Q 1Y0 <-> Data Pointer/QCurrentSetPoints[9]
//     Term 18 (APS4322-7000)/APS Outputs/Current Q 1Y1 <-> Data Pointer/QCurrentSetPoints[10]
//     Term 18 (APS4322-7000)/APS Outputs/Current Q 1Y2 <-> Data Pointer/QCurrentSetPoints[11]
//     Term 18 (APS4322-7000)/APS Outputs/Current Q 2Y0 <-> Data Pointer/QCurrentSetPoints[15]
//     Term 18 (APS4322-7000)/APS Outputs/Current Q 2Y1 <-> Data Pointer/QCurrentSetPoints[16]
//     Term 18 (APS4322-7000)/APS Outputs/Current Q 2Y2 <-> Data Pointer/QCurrentSetPoints[17]
//     Term 18 (APS4322-7000)/APS Outputs/Current Q 3Y0 <-> Data Pointer/QCurrentSetPoints[21]
//     Term 18 (APS4322-7000)/APS Outputs/Current Q 3Y1 <-> Data Pointer/QCurrentSetPoints[22]
//     Term 18 (APS4322-7000)/APS Outputs/Current Q 3Y2 <-> Data Pointer/QCurrentSetPoints[23]
//     Term 18 (APS4322-7000)/APS Outputs/PhiE 0X0 <-> Data Pointer/PhiSetPoints[0]
//     Term 18 (APS4322-7000)/APS Outputs/PhiE 0X1 <-> Data Pointer/PhiSetPoints[1]
//     Term 18 (APS4322-7000)/APS Outputs/PhiE 0X2 <-> Data Pointer/PhiSetPoints[2]
//     Term 18 (APS4322-7000)/APS Outputs/PhiE 1X0 <-> Data Pointer/PhiSetPoints[6]
//     Term 18 (APS4322-7000)/APS Outputs/PhiE 1X1 <-> Data Pointer/PhiSetPoints[7]
//     Term 18 (APS4322-7000)/APS Outputs/PhiE 1X2 <-> Data Pointer/PhiSetPoints[8]
//     Term 18 (APS4322-7000)/APS Outputs/PhiE 2X0 <-> Data Pointer/PhiSetPoints[12]
//     Term 18 (APS4322-7000)/APS Outputs/PhiE 2X1 <-> Data Pointer/PhiSetPoints[13]
//     Term 18 (APS4322-7000)/APS Outputs/PhiE 2X2 <-> Data Pointer/PhiSetPoints[14]
//     Term 18 (APS4322-7000)/APS Outputs/PhiE 3X0 <-> Data Pointer/PhiSetPoints[18]
//     Term 18 (APS4322-7000)/APS Outputs/PhiE 3X1 <-> Data Pointer/PhiSetPoints[19]
//     Term 18 (APS4322-7000)/APS Outputs/PhiE 3X2 <-> Data Pointer/PhiSetPoints[20]
//     Term 18 (APS4322-7000)/APS Outputs/PhiE 0Y0 <-> Data Pointer/PhiSetPoints[3]
//     Term 18 (APS4322-7000)/APS Outputs/PhiE 0Y1 <-> Data Pointer/PhiSetPoints[4]
//     Term 18 (APS4322-7000)/APS Outputs/PhiE 0Y2 <-> Data Pointer/PhiSetPoints[5]
//     Term 18 (APS4322-7000)/APS Outputs/PhiE 1Y0 <-> Data Pointer/PhiSetPoints[9]
//     Term 18 (APS4322-7000)/APS Outputs/PhiE 1Y1 <-> Data Pointer/PhiSetPoints[10]
//     Term 18 (APS4322-7000)/APS Outputs/PhiE 1Y2 <-> Data Pointer/PhiSetPoints[11]
//     Term 18 (APS4322-7000)/APS Outputs/PhiE 2Y0 <-> Data Pointer/PhiSetPoints[15]
//     Term 18 (APS4322-7000)/APS Outputs/PhiE 2Y1 <-> Data Pointer/PhiSetPoints[16]
//     Term 18 (APS4322-7000)/APS Outputs/PhiE 2Y2 <-> Data Pointer/PhiSetPoints[17]
//     Term 18 (APS4322-7000)/APS Outputs/PhiE 3Y0 <-> Data Pointer/PhiSetPoints[21]
//     Term 18 (APS4322-7000)/APS Outputs/PhiE 3Y1 <-> Data Pointer/PhiSetPoints[22]
//     Term 18 (APS4322-7000)/APS Outputs/PhiE 3Y2 <-> Data Pointer/PhiSetPoints[23]
//     Term 18 (APS4322-7000)/Term 19 (APS4322-5000)/FB Inputs/A{0..8 step 2} X-Field <-> Data Pointer/HallSensorFieldsXYZ[{0..12 step 3}]  (5 links)
//     Term 18 (APS4322-7000)/Term 19 (APS4322-5000)/FB Inputs/A{0..8 step 2} Y-Field <-> Data Pointer/HallSensorFieldsXYZ[{1..13 step 3}]  (5 links)
//     Term 18 (APS4322-7000)/Term 19 (APS4322-5000)/FB Inputs/A{0..8 step 2} Z-Field <-> Data Pointer/HallSensorFieldsXYZ[{2..14 step 3}]  (5 links)
//     Term 18 (APS4322-7000)/Term 19 (APS4322-5000)/FB Inputs/B{1..9 step 2} X-Field <-> Data Pointer/HallSensorFieldsXYZ[{15..27 step 3}]  (5 links)
//     Term 18 (APS4322-7000)/Term 19 (APS4322-5000)/FB Inputs/B{1..9 step 2} Y-Field <-> Data Pointer/HallSensorFieldsXYZ[{16..28 step 3}]  (5 links)
//     Term 18 (APS4322-7000)/Term 19 (APS4322-5000)/FB Inputs/B{1..9 step 2} Z-Field <-> Data Pointer/HallSensorFieldsXYZ[{17..29 step 3}]  (5 links)
//     Term 18 (APS4322-7000)/Term 19 (APS4322-5000)/FB Inputs/C{0..8 step 2} X-Field <-> Data Pointer/HallSensorFieldsXYZ[{30..42 step 3}]  (5 links)
//     Term 18 (APS4322-7000)/Term 19 (APS4322-5000)/FB Inputs/C{0..8 step 2} Y-Field <-> Data Pointer/HallSensorFieldsXYZ[{31..43 step 3}]  (5 links)
//     Term 18 (APS4322-7000)/Term 19 (APS4322-5000)/FB Inputs/C{0..8 step 2} Z-Field <-> Data Pointer/HallSensorFieldsXYZ[{32..44 step 3}]  (5 links)
//     Term 18 (APS4322-7000)/Term 19 (APS4322-5000)/FB Inputs/D{1..9 step 2} X-Field <-> Data Pointer/HallSensorFieldsXYZ[{45..57 step 3}]  (5 links)
//     Term 18 (APS4322-7000)/Term 19 (APS4322-5000)/FB Inputs/D{1..9 step 2} Y-Field <-> Data Pointer/HallSensorFieldsXYZ[{46..58 step 3}]  (5 links)
//     Term 18 (APS4322-7000)/Term 19 (APS4322-5000)/FB Inputs/D{1..9 step 2} Z-Field <-> Data Pointer/HallSensorFieldsXYZ[{47..59 step 3}]  (5 links)
//     Term 18 (APS4322-7000)/Term 19 (APS4322-5000)/FB Inputs/E{0..8 step 2} X-Field <-> Data Pointer/HallSensorFieldsXYZ[{60..72 step 3}]  (5 links)
//     Term 18 (APS4322-7000)/Term 19 (APS4322-5000)/FB Inputs/E{0..8 step 2} Y-Field <-> Data Pointer/HallSensorFieldsXYZ[{61..73 step 3}]  (5 links)
//     Term 18 (APS4322-7000)/Term 19 (APS4322-5000)/FB Inputs/E{0..8 step 2} Z-Field <-> Data Pointer/HallSensorFieldsXYZ[{62..74 step 3}]  (5 links)
//     Term 18 (APS4322-7000)/Term 19 (APS4322-5000)/FB Inputs/F{1..9 step 2} X-Field <-> Data Pointer/HallSensorFieldsXYZ[{75..87 step 3}]  (5 links)
//     Term 18 (APS4322-7000)/Term 19 (APS4322-5000)/FB Inputs/F{1..9 step 2} Y-Field <-> Data Pointer/HallSensorFieldsXYZ[{76..88 step 3}]  (5 links)
//     Term 18 (APS4322-7000)/Term 19 (APS4322-5000)/FB Inputs/F{1..9 step 2} Z-Field <-> Data Pointer/HallSensorFieldsXYZ[{77..89 step 3}]  (5 links)
//     Term 18 (APS4322-7000)/Term 19 (APS4322-5000)/FB Inputs/G{0..8 step 2} X-Field <-> Data Pointer/HallSensorFieldsXYZ[{90..102 step 3}]  (5 links)
//     Term 18 (APS4322-7000)/Term 19 (APS4322-5000)/FB Inputs/G{0..8 step 2} Y-Field <-> Data Pointer/HallSensorFieldsXYZ[{91..103 step 3}]  (5 links)
//     Term 18 (APS4322-7000)/Term 19 (APS4322-5000)/FB Inputs/G{0..8 step 2} Z-Field <-> Data Pointer/HallSensorFieldsXYZ[{92..104 step 3}]  (5 links)
//     Term 18 (APS4322-7000)/Term 19 (APS4322-5000)/FB Inputs/H{1..9 step 2} X-Field <-> Data Pointer/HallSensorFieldsXYZ[{105..117 step 3}]  (5 links)
//     Term 18 (APS4322-7000)/Term 19 (APS4322-5000)/FB Inputs/H{1..9 step 2} Y-Field <-> Data Pointer/HallSensorFieldsXYZ[{106..118 step 3}]  (5 links)
//     Term 18 (APS4322-7000)/Term 19 (APS4322-5000)/FB Inputs/H{1..9 step 2} Z-Field <-> Data Pointer/HallSensorFieldsXYZ[{107..119 step 3}]  (5 links)
//     Term 18 (APS4322-7000)/Term 19 (APS4322-5000)/FB Inputs/I{0..8 step 2} X-Field <-> Data Pointer/HallSensorFieldsXYZ[{120..132 step 3}]  (5 links)
//     Term 18 (APS4322-7000)/Term 19 (APS4322-5000)/FB Inputs/I{0..8 step 2} Y-Field <-> Data Pointer/HallSensorFieldsXYZ[{121..133 step 3}]  (5 links)
//     Term 18 (APS4322-7000)/Term 19 (APS4322-5000)/FB Inputs/I{0..8 step 2} Z-Field <-> Data Pointer/HallSensorFieldsXYZ[{122..134 step 3}]  (5 links)
//     Term 18 (APS4322-7000)/Term 19 (APS4322-5000)/FB Inputs/J{1..9 step 2} X-Field <-> Data Pointer/HallSensorFieldsXYZ[{135..147 step 3}]  (5 links)
//     Term 18 (APS4322-7000)/Term 19 (APS4322-5000)/FB Inputs/J{1..9 step 2} Y-Field <-> Data Pointer/HallSensorFieldsXYZ[{136..148 step 3}]  (5 links)
//     Term 18 (APS4322-7000)/Term 19 (APS4322-5000)/FB Inputs/J{1..9 step 2} Z-Field <-> Data Pointer/HallSensorFieldsXYZ[{137..149 step 3}]  (5 links)
//     Term 18 (APS4322-7000)/Term 19 (APS4322-5000)/FB Inputs/Status <-> Data Pointer/FeedbackStatus
//   Device 5 (EtherCAT) <-> TcCOM Objects/XPlanar/Part1/APS4322_P1_4
//     Term 12 (APS4322-7000)/APS Comm Inputs/CommStatusWord <-> Data Pointer/MoverCommStatusWord
//     Term 12 (APS4322-7000)/APS Comm Inputs/Data {1..4} <-> Data Pointer/MoverCommDataIn[{0..3}]  (4 links)
//     Term 12 (APS4322-7000)/APS Comm Outputs/CommControlWord <-> Data Pointer/MoverCommControlWord
//     Term 12 (APS4322-7000)/APS Comm Outputs/Data 1 <-> Data Pointer/MoverCommDataOut
//     Term 12 (APS4322-7000)/APS Diagdata/DC Link Voltage <-> Data Pointer/DcLinkVoltage
//     Term 12 (APS4322-7000)/APS Diagdata/Power supply current <-> Data Pointer/PowerSupplyCurrent
//     Term 12 (APS4322-7000)/APS Inputs/StatusWord <-> Data Pointer/PowerUnitStatusWord
//     Term 12 (APS4322-7000)/APS Outputs/ControlWord <-> Data Pointer/PowerUnitControlWord
//     Term 12 (APS4322-7000)/APS Outputs/Current D 0X0 <-> Data Pointer/DCurrentSetPoints[0]
//     Term 12 (APS4322-7000)/APS Outputs/Current D 0X1 <-> Data Pointer/DCurrentSetPoints[1]
//     Term 12 (APS4322-7000)/APS Outputs/Current D 0X2 <-> Data Pointer/DCurrentSetPoints[2]
//     Term 12 (APS4322-7000)/APS Outputs/Current D 1X0 <-> Data Pointer/DCurrentSetPoints[6]
//     Term 12 (APS4322-7000)/APS Outputs/Current D 1X1 <-> Data Pointer/DCurrentSetPoints[7]
//     Term 12 (APS4322-7000)/APS Outputs/Current D 1X2 <-> Data Pointer/DCurrentSetPoints[8]
//     Term 12 (APS4322-7000)/APS Outputs/Current D 2X0 <-> Data Pointer/DCurrentSetPoints[12]
//     Term 12 (APS4322-7000)/APS Outputs/Current D 2X1 <-> Data Pointer/DCurrentSetPoints[13]
//     Term 12 (APS4322-7000)/APS Outputs/Current D 2X2 <-> Data Pointer/DCurrentSetPoints[14]
//     Term 12 (APS4322-7000)/APS Outputs/Current D 3X0 <-> Data Pointer/DCurrentSetPoints[18]
//     Term 12 (APS4322-7000)/APS Outputs/Current D 3X1 <-> Data Pointer/DCurrentSetPoints[19]
//     Term 12 (APS4322-7000)/APS Outputs/Current D 3X2 <-> Data Pointer/DCurrentSetPoints[20]
//     Term 12 (APS4322-7000)/APS Outputs/Current D 0Y0 <-> Data Pointer/DCurrentSetPoints[3]
//     Term 12 (APS4322-7000)/APS Outputs/Current D 0Y1 <-> Data Pointer/DCurrentSetPoints[4]
//     Term 12 (APS4322-7000)/APS Outputs/Current D 0Y2 <-> Data Pointer/DCurrentSetPoints[5]
//     Term 12 (APS4322-7000)/APS Outputs/Current D 1Y0 <-> Data Pointer/DCurrentSetPoints[9]
//     Term 12 (APS4322-7000)/APS Outputs/Current D 1Y1 <-> Data Pointer/DCurrentSetPoints[10]
//     Term 12 (APS4322-7000)/APS Outputs/Current D 1Y2 <-> Data Pointer/DCurrentSetPoints[11]
//     Term 12 (APS4322-7000)/APS Outputs/Current D 2Y0 <-> Data Pointer/DCurrentSetPoints[15]
//     Term 12 (APS4322-7000)/APS Outputs/Current D 2Y1 <-> Data Pointer/DCurrentSetPoints[16]
//     Term 12 (APS4322-7000)/APS Outputs/Current D 2Y2 <-> Data Pointer/DCurrentSetPoints[17]
//     Term 12 (APS4322-7000)/APS Outputs/Current D 3Y0 <-> Data Pointer/DCurrentSetPoints[21]
//     Term 12 (APS4322-7000)/APS Outputs/Current D 3Y1 <-> Data Pointer/DCurrentSetPoints[22]
//     Term 12 (APS4322-7000)/APS Outputs/Current D 3Y2 <-> Data Pointer/DCurrentSetPoints[23]
//     Term 12 (APS4322-7000)/APS Outputs/Current Q 0X0 <-> Data Pointer/QCurrentSetPoints[0]
//     Term 12 (APS4322-7000)/APS Outputs/Current Q 0X1 <-> Data Pointer/QCurrentSetPoints[1]
//     Term 12 (APS4322-7000)/APS Outputs/Current Q 0X2 <-> Data Pointer/QCurrentSetPoints[2]
//     Term 12 (APS4322-7000)/APS Outputs/Current Q 1X0 <-> Data Pointer/QCurrentSetPoints[6]
//     Term 12 (APS4322-7000)/APS Outputs/Current Q 1X1 <-> Data Pointer/QCurrentSetPoints[7]
//     Term 12 (APS4322-7000)/APS Outputs/Current Q 1X2 <-> Data Pointer/QCurrentSetPoints[8]
//     Term 12 (APS4322-7000)/APS Outputs/Current Q 2X0 <-> Data Pointer/QCurrentSetPoints[12]
//     Term 12 (APS4322-7000)/APS Outputs/Current Q 2X1 <-> Data Pointer/QCurrentSetPoints[13]
//     Term 12 (APS4322-7000)/APS Outputs/Current Q 2X2 <-> Data Pointer/QCurrentSetPoints[14]
//     Term 12 (APS4322-7000)/APS Outputs/Current Q 3X0 <-> Data Pointer/QCurrentSetPoints[18]
//     Term 12 (APS4322-7000)/APS Outputs/Current Q 3X1 <-> Data Pointer/QCurrentSetPoints[19]
//     Term 12 (APS4322-7000)/APS Outputs/Current Q 3X2 <-> Data Pointer/QCurrentSetPoints[20]
//     Term 12 (APS4322-7000)/APS Outputs/Current Q 0Y0 <-> Data Pointer/QCurrentSetPoints[3]
//     Term 12 (APS4322-7000)/APS Outputs/Current Q 0Y1 <-> Data Pointer/QCurrentSetPoints[4]
//     Term 12 (APS4322-7000)/APS Outputs/Current Q 0Y2 <-> Data Pointer/QCurrentSetPoints[5]
//     Term 12 (APS4322-7000)/APS Outputs/Current Q 1Y0 <-> Data Pointer/QCurrentSetPoints[9]
//     Term 12 (APS4322-7000)/APS Outputs/Current Q 1Y1 <-> Data Pointer/QCurrentSetPoints[10]
//     Term 12 (APS4322-7000)/APS Outputs/Current Q 1Y2 <-> Data Pointer/QCurrentSetPoints[11]
//     Term 12 (APS4322-7000)/APS Outputs/Current Q 2Y0 <-> Data Pointer/QCurrentSetPoints[15]
//     Term 12 (APS4322-7000)/APS Outputs/Current Q 2Y1 <-> Data Pointer/QCurrentSetPoints[16]
//     Term 12 (APS4322-7000)/APS Outputs/Current Q 2Y2 <-> Data Pointer/QCurrentSetPoints[17]
//     Term 12 (APS4322-7000)/APS Outputs/Current Q 3Y0 <-> Data Pointer/QCurrentSetPoints[21]
//     Term 12 (APS4322-7000)/APS Outputs/Current Q 3Y1 <-> Data Pointer/QCurrentSetPoints[22]
//     Term 12 (APS4322-7000)/APS Outputs/Current Q 3Y2 <-> Data Pointer/QCurrentSetPoints[23]
//     Term 12 (APS4322-7000)/APS Outputs/PhiE 0X0 <-> Data Pointer/PhiSetPoints[0]
//     Term 12 (APS4322-7000)/APS Outputs/PhiE 0X1 <-> Data Pointer/PhiSetPoints[1]
//     Term 12 (APS4322-7000)/APS Outputs/PhiE 0X2 <-> Data Pointer/PhiSetPoints[2]
//     Term 12 (APS4322-7000)/APS Outputs/PhiE 1X0 <-> Data Pointer/PhiSetPoints[6]
//     Term 12 (APS4322-7000)/APS Outputs/PhiE 1X1 <-> Data Pointer/PhiSetPoints[7]
//     Term 12 (APS4322-7000)/APS Outputs/PhiE 1X2 <-> Data Pointer/PhiSetPoints[8]
//     Term 12 (APS4322-7000)/APS Outputs/PhiE 2X0 <-> Data Pointer/PhiSetPoints[12]
//     Term 12 (APS4322-7000)/APS Outputs/PhiE 2X1 <-> Data Pointer/PhiSetPoints[13]
//     Term 12 (APS4322-7000)/APS Outputs/PhiE 2X2 <-> Data Pointer/PhiSetPoints[14]
//     Term 12 (APS4322-7000)/APS Outputs/PhiE 3X0 <-> Data Pointer/PhiSetPoints[18]
//     Term 12 (APS4322-7000)/APS Outputs/PhiE 3X1 <-> Data Pointer/PhiSetPoints[19]
//     Term 12 (APS4322-7000)/APS Outputs/PhiE 3X2 <-> Data Pointer/PhiSetPoints[20]
//     Term 12 (APS4322-7000)/APS Outputs/PhiE 0Y0 <-> Data Pointer/PhiSetPoints[3]
//     Term 12 (APS4322-7000)/APS Outputs/PhiE 0Y1 <-> Data Pointer/PhiSetPoints[4]
//     Term 12 (APS4322-7000)/APS Outputs/PhiE 0Y2 <-> Data Pointer/PhiSetPoints[5]
//     Term 12 (APS4322-7000)/APS Outputs/PhiE 1Y0 <-> Data Pointer/PhiSetPoints[9]
//     Term 12 (APS4322-7000)/APS Outputs/PhiE 1Y1 <-> Data Pointer/PhiSetPoints[10]
//     Term 12 (APS4322-7000)/APS Outputs/PhiE 1Y2 <-> Data Pointer/PhiSetPoints[11]
//     Term 12 (APS4322-7000)/APS Outputs/PhiE 2Y0 <-> Data Pointer/PhiSetPoints[15]
//     Term 12 (APS4322-7000)/APS Outputs/PhiE 2Y1 <-> Data Pointer/PhiSetPoints[16]
//     Term 12 (APS4322-7000)/APS Outputs/PhiE 2Y2 <-> Data Pointer/PhiSetPoints[17]
//     Term 12 (APS4322-7000)/APS Outputs/PhiE 3Y0 <-> Data Pointer/PhiSetPoints[21]
//     Term 12 (APS4322-7000)/APS Outputs/PhiE 3Y1 <-> Data Pointer/PhiSetPoints[22]
//     Term 12 (APS4322-7000)/APS Outputs/PhiE 3Y2 <-> Data Pointer/PhiSetPoints[23]
//     Term 12 (APS4322-7000)/Term 13 (APS4322-5000)/FB Inputs/A{0..8 step 2} X-Field <-> Data Pointer/HallSensorFieldsXYZ[{0..12 step 3}]  (5 links)
//     Term 12 (APS4322-7000)/Term 13 (APS4322-5000)/FB Inputs/A{0..8 step 2} Y-Field <-> Data Pointer/HallSensorFieldsXYZ[{1..13 step 3}]  (5 links)
//     Term 12 (APS4322-7000)/Term 13 (APS4322-5000)/FB Inputs/A{0..8 step 2} Z-Field <-> Data Pointer/HallSensorFieldsXYZ[{2..14 step 3}]  (5 links)
//     Term 12 (APS4322-7000)/Term 13 (APS4322-5000)/FB Inputs/B{1..9 step 2} X-Field <-> Data Pointer/HallSensorFieldsXYZ[{15..27 step 3}]  (5 links)
//     Term 12 (APS4322-7000)/Term 13 (APS4322-5000)/FB Inputs/B{1..9 step 2} Y-Field <-> Data Pointer/HallSensorFieldsXYZ[{16..28 step 3}]  (5 links)
//     Term 12 (APS4322-7000)/Term 13 (APS4322-5000)/FB Inputs/B{1..9 step 2} Z-Field <-> Data Pointer/HallSensorFieldsXYZ[{17..29 step 3}]  (5 links)
//     Term 12 (APS4322-7000)/Term 13 (APS4322-5000)/FB Inputs/C{0..8 step 2} X-Field <-> Data Pointer/HallSensorFieldsXYZ[{30..42 step 3}]  (5 links)
//     Term 12 (APS4322-7000)/Term 13 (APS4322-5000)/FB Inputs/C{0..8 step 2} Y-Field <-> Data Pointer/HallSensorFieldsXYZ[{31..43 step 3}]  (5 links)
//     Term 12 (APS4322-7000)/Term 13 (APS4322-5000)/FB Inputs/C{0..8 step 2} Z-Field <-> Data Pointer/HallSensorFieldsXYZ[{32..44 step 3}]  (5 links)
//     Term 12 (APS4322-7000)/Term 13 (APS4322-5000)/FB Inputs/D{1..9 step 2} X-Field <-> Data Pointer/HallSensorFieldsXYZ[{45..57 step 3}]  (5 links)
//     Term 12 (APS4322-7000)/Term 13 (APS4322-5000)/FB Inputs/D{1..9 step 2} Y-Field <-> Data Pointer/HallSensorFieldsXYZ[{46..58 step 3}]  (5 links)
//     Term 12 (APS4322-7000)/Term 13 (APS4322-5000)/FB Inputs/D{1..9 step 2} Z-Field <-> Data Pointer/HallSensorFieldsXYZ[{47..59 step 3}]  (5 links)
//     Term 12 (APS4322-7000)/Term 13 (APS4322-5000)/FB Inputs/E{0..8 step 2} X-Field <-> Data Pointer/HallSensorFieldsXYZ[{60..72 step 3}]  (5 links)
//     Term 12 (APS4322-7000)/Term 13 (APS4322-5000)/FB Inputs/E{0..8 step 2} Y-Field <-> Data Pointer/HallSensorFieldsXYZ[{61..73 step 3}]  (5 links)
//     Term 12 (APS4322-7000)/Term 13 (APS4322-5000)/FB Inputs/E{0..8 step 2} Z-Field <-> Data Pointer/HallSensorFieldsXYZ[{62..74 step 3}]  (5 links)
//     Term 12 (APS4322-7000)/Term 13 (APS4322-5000)/FB Inputs/F{1..9 step 2} X-Field <-> Data Pointer/HallSensorFieldsXYZ[{75..87 step 3}]  (5 links)
//     Term 12 (APS4322-7000)/Term 13 (APS4322-5000)/FB Inputs/F{1..9 step 2} Y-Field <-> Data Pointer/HallSensorFieldsXYZ[{76..88 step 3}]  (5 links)
//     Term 12 (APS4322-7000)/Term 13 (APS4322-5000)/FB Inputs/F{1..9 step 2} Z-Field <-> Data Pointer/HallSensorFieldsXYZ[{77..89 step 3}]  (5 links)
//     Term 12 (APS4322-7000)/Term 13 (APS4322-5000)/FB Inputs/G{0..8 step 2} X-Field <-> Data Pointer/HallSensorFieldsXYZ[{90..102 step 3}]  (5 links)
//     Term 12 (APS4322-7000)/Term 13 (APS4322-5000)/FB Inputs/G{0..8 step 2} Y-Field <-> Data Pointer/HallSensorFieldsXYZ[{91..103 step 3}]  (5 links)
//     Term 12 (APS4322-7000)/Term 13 (APS4322-5000)/FB Inputs/G{0..8 step 2} Z-Field <-> Data Pointer/HallSensorFieldsXYZ[{92..104 step 3}]  (5 links)
//     Term 12 (APS4322-7000)/Term 13 (APS4322-5000)/FB Inputs/H{1..9 step 2} X-Field <-> Data Pointer/HallSensorFieldsXYZ[{105..117 step 3}]  (5 links)
//     Term 12 (APS4322-7000)/Term 13 (APS4322-5000)/FB Inputs/H{1..9 step 2} Y-Field <-> Data Pointer/HallSensorFieldsXYZ[{106..118 step 3}]  (5 links)
//     Term 12 (APS4322-7000)/Term 13 (APS4322-5000)/FB Inputs/H{1..9 step 2} Z-Field <-> Data Pointer/HallSensorFieldsXYZ[{107..119 step 3}]  (5 links)
//     Term 12 (APS4322-7000)/Term 13 (APS4322-5000)/FB Inputs/I{0..8 step 2} X-Field <-> Data Pointer/HallSensorFieldsXYZ[{120..132 step 3}]  (5 links)
//     Term 12 (APS4322-7000)/Term 13 (APS4322-5000)/FB Inputs/I{0..8 step 2} Y-Field <-> Data Pointer/HallSensorFieldsXYZ[{121..133 step 3}]  (5 links)
//     Term 12 (APS4322-7000)/Term 13 (APS4322-5000)/FB Inputs/I{0..8 step 2} Z-Field <-> Data Pointer/HallSensorFieldsXYZ[{122..134 step 3}]  (5 links)
//     Term 12 (APS4322-7000)/Term 13 (APS4322-5000)/FB Inputs/J{1..9 step 2} X-Field <-> Data Pointer/HallSensorFieldsXYZ[{135..147 step 3}]  (5 links)
//     Term 12 (APS4322-7000)/Term 13 (APS4322-5000)/FB Inputs/J{1..9 step 2} Y-Field <-> Data Pointer/HallSensorFieldsXYZ[{136..148 step 3}]  (5 links)
//     Term 12 (APS4322-7000)/Term 13 (APS4322-5000)/FB Inputs/J{1..9 step 2} Z-Field <-> Data Pointer/HallSensorFieldsXYZ[{137..149 step 3}]  (5 links)
//     Term 12 (APS4322-7000)/Term 13 (APS4322-5000)/FB Inputs/Status <-> Data Pointer/FeedbackStatus
//   Device 5 (EtherCAT) <-> TcCOM Objects/XPlanar/Part1/APS4322_P1_5
//     Term 10 (APS4322-7000)/APS Comm Inputs/CommStatusWord <-> Data Pointer/MoverCommStatusWord
//     Term 10 (APS4322-7000)/APS Comm Inputs/Data {1..4} <-> Data Pointer/MoverCommDataIn[{0..3}]  (4 links)
//     Term 10 (APS4322-7000)/APS Comm Outputs/CommControlWord <-> Data Pointer/MoverCommControlWord
//     Term 10 (APS4322-7000)/APS Comm Outputs/Data 1 <-> Data Pointer/MoverCommDataOut
//     Term 10 (APS4322-7000)/APS Diagdata/DC Link Voltage <-> Data Pointer/DcLinkVoltage
//     Term 10 (APS4322-7000)/APS Diagdata/Power supply current <-> Data Pointer/PowerSupplyCurrent
//     Term 10 (APS4322-7000)/APS Inputs/StatusWord <-> Data Pointer/PowerUnitStatusWord
//     Term 10 (APS4322-7000)/APS Outputs/ControlWord <-> Data Pointer/PowerUnitControlWord
//     Term 10 (APS4322-7000)/APS Outputs/Current D 0X0 <-> Data Pointer/DCurrentSetPoints[0]
//     Term 10 (APS4322-7000)/APS Outputs/Current D 0X1 <-> Data Pointer/DCurrentSetPoints[1]
//     Term 10 (APS4322-7000)/APS Outputs/Current D 0X2 <-> Data Pointer/DCurrentSetPoints[2]
//     Term 10 (APS4322-7000)/APS Outputs/Current D 1X0 <-> Data Pointer/DCurrentSetPoints[6]
//     Term 10 (APS4322-7000)/APS Outputs/Current D 1X1 <-> Data Pointer/DCurrentSetPoints[7]
//     Term 10 (APS4322-7000)/APS Outputs/Current D 1X2 <-> Data Pointer/DCurrentSetPoints[8]
//     Term 10 (APS4322-7000)/APS Outputs/Current D 2X0 <-> Data Pointer/DCurrentSetPoints[12]
//     Term 10 (APS4322-7000)/APS Outputs/Current D 2X1 <-> Data Pointer/DCurrentSetPoints[13]
//     Term 10 (APS4322-7000)/APS Outputs/Current D 2X2 <-> Data Pointer/DCurrentSetPoints[14]
//     Term 10 (APS4322-7000)/APS Outputs/Current D 3X0 <-> Data Pointer/DCurrentSetPoints[18]
//     Term 10 (APS4322-7000)/APS Outputs/Current D 3X1 <-> Data Pointer/DCurrentSetPoints[19]
//     Term 10 (APS4322-7000)/APS Outputs/Current D 3X2 <-> Data Pointer/DCurrentSetPoints[20]
//     Term 10 (APS4322-7000)/APS Outputs/Current D 0Y0 <-> Data Pointer/DCurrentSetPoints[3]
//     Term 10 (APS4322-7000)/APS Outputs/Current D 0Y1 <-> Data Pointer/DCurrentSetPoints[4]
//     Term 10 (APS4322-7000)/APS Outputs/Current D 0Y2 <-> Data Pointer/DCurrentSetPoints[5]
//     Term 10 (APS4322-7000)/APS Outputs/Current D 1Y0 <-> Data Pointer/DCurrentSetPoints[9]
//     Term 10 (APS4322-7000)/APS Outputs/Current D 1Y1 <-> Data Pointer/DCurrentSetPoints[10]
//     Term 10 (APS4322-7000)/APS Outputs/Current D 1Y2 <-> Data Pointer/DCurrentSetPoints[11]
//     Term 10 (APS4322-7000)/APS Outputs/Current D 2Y0 <-> Data Pointer/DCurrentSetPoints[15]
//     Term 10 (APS4322-7000)/APS Outputs/Current D 2Y1 <-> Data Pointer/DCurrentSetPoints[16]
//     Term 10 (APS4322-7000)/APS Outputs/Current D 2Y2 <-> Data Pointer/DCurrentSetPoints[17]
//     Term 10 (APS4322-7000)/APS Outputs/Current D 3Y0 <-> Data Pointer/DCurrentSetPoints[21]
//     Term 10 (APS4322-7000)/APS Outputs/Current D 3Y1 <-> Data Pointer/DCurrentSetPoints[22]
//     Term 10 (APS4322-7000)/APS Outputs/Current D 3Y2 <-> Data Pointer/DCurrentSetPoints[23]
//     Term 10 (APS4322-7000)/APS Outputs/Current Q 0X0 <-> Data Pointer/QCurrentSetPoints[0]
//     Term 10 (APS4322-7000)/APS Outputs/Current Q 0X1 <-> Data Pointer/QCurrentSetPoints[1]
//     Term 10 (APS4322-7000)/APS Outputs/Current Q 0X2 <-> Data Pointer/QCurrentSetPoints[2]
//     Term 10 (APS4322-7000)/APS Outputs/Current Q 1X0 <-> Data Pointer/QCurrentSetPoints[6]
//     Term 10 (APS4322-7000)/APS Outputs/Current Q 1X1 <-> Data Pointer/QCurrentSetPoints[7]
//     Term 10 (APS4322-7000)/APS Outputs/Current Q 1X2 <-> Data Pointer/QCurrentSetPoints[8]
//     Term 10 (APS4322-7000)/APS Outputs/Current Q 2X0 <-> Data Pointer/QCurrentSetPoints[12]
//     Term 10 (APS4322-7000)/APS Outputs/Current Q 2X1 <-> Data Pointer/QCurrentSetPoints[13]
//     Term 10 (APS4322-7000)/APS Outputs/Current Q 2X2 <-> Data Pointer/QCurrentSetPoints[14]
//     Term 10 (APS4322-7000)/APS Outputs/Current Q 3X0 <-> Data Pointer/QCurrentSetPoints[18]
//     Term 10 (APS4322-7000)/APS Outputs/Current Q 3X1 <-> Data Pointer/QCurrentSetPoints[19]
//     Term 10 (APS4322-7000)/APS Outputs/Current Q 3X2 <-> Data Pointer/QCurrentSetPoints[20]
//     Term 10 (APS4322-7000)/APS Outputs/Current Q 0Y0 <-> Data Pointer/QCurrentSetPoints[3]
//     Term 10 (APS4322-7000)/APS Outputs/Current Q 0Y1 <-> Data Pointer/QCurrentSetPoints[4]
//     Term 10 (APS4322-7000)/APS Outputs/Current Q 0Y2 <-> Data Pointer/QCurrentSetPoints[5]
//     Term 10 (APS4322-7000)/APS Outputs/Current Q 1Y0 <-> Data Pointer/QCurrentSetPoints[9]
//     Term 10 (APS4322-7000)/APS Outputs/Current Q 1Y1 <-> Data Pointer/QCurrentSetPoints[10]
//     Term 10 (APS4322-7000)/APS Outputs/Current Q 1Y2 <-> Data Pointer/QCurrentSetPoints[11]
//     Term 10 (APS4322-7000)/APS Outputs/Current Q 2Y0 <-> Data Pointer/QCurrentSetPoints[15]
//     Term 10 (APS4322-7000)/APS Outputs/Current Q 2Y1 <-> Data Pointer/QCurrentSetPoints[16]
//     Term 10 (APS4322-7000)/APS Outputs/Current Q 2Y2 <-> Data Pointer/QCurrentSetPoints[17]
//     Term 10 (APS4322-7000)/APS Outputs/Current Q 3Y0 <-> Data Pointer/QCurrentSetPoints[21]
//     Term 10 (APS4322-7000)/APS Outputs/Current Q 3Y1 <-> Data Pointer/QCurrentSetPoints[22]
//     Term 10 (APS4322-7000)/APS Outputs/Current Q 3Y2 <-> Data Pointer/QCurrentSetPoints[23]
//     Term 10 (APS4322-7000)/APS Outputs/PhiE 0X0 <-> Data Pointer/PhiSetPoints[0]
//     Term 10 (APS4322-7000)/APS Outputs/PhiE 0X1 <-> Data Pointer/PhiSetPoints[1]
//     Term 10 (APS4322-7000)/APS Outputs/PhiE 0X2 <-> Data Pointer/PhiSetPoints[2]
//     Term 10 (APS4322-7000)/APS Outputs/PhiE 1X0 <-> Data Pointer/PhiSetPoints[6]
//     Term 10 (APS4322-7000)/APS Outputs/PhiE 1X1 <-> Data Pointer/PhiSetPoints[7]
//     Term 10 (APS4322-7000)/APS Outputs/PhiE 1X2 <-> Data Pointer/PhiSetPoints[8]
//     Term 10 (APS4322-7000)/APS Outputs/PhiE 2X0 <-> Data Pointer/PhiSetPoints[12]
//     Term 10 (APS4322-7000)/APS Outputs/PhiE 2X1 <-> Data Pointer/PhiSetPoints[13]
//     Term 10 (APS4322-7000)/APS Outputs/PhiE 2X2 <-> Data Pointer/PhiSetPoints[14]
//     Term 10 (APS4322-7000)/APS Outputs/PhiE 3X0 <-> Data Pointer/PhiSetPoints[18]
//     Term 10 (APS4322-7000)/APS Outputs/PhiE 3X1 <-> Data Pointer/PhiSetPoints[19]
//     Term 10 (APS4322-7000)/APS Outputs/PhiE 3X2 <-> Data Pointer/PhiSetPoints[20]
//     Term 10 (APS4322-7000)/APS Outputs/PhiE 0Y0 <-> Data Pointer/PhiSetPoints[3]
//     Term 10 (APS4322-7000)/APS Outputs/PhiE 0Y1 <-> Data Pointer/PhiSetPoints[4]
//     Term 10 (APS4322-7000)/APS Outputs/PhiE 0Y2 <-> Data Pointer/PhiSetPoints[5]
//     Term 10 (APS4322-7000)/APS Outputs/PhiE 1Y0 <-> Data Pointer/PhiSetPoints[9]
//     Term 10 (APS4322-7000)/APS Outputs/PhiE 1Y1 <-> Data Pointer/PhiSetPoints[10]
//     Term 10 (APS4322-7000)/APS Outputs/PhiE 1Y2 <-> Data Pointer/PhiSetPoints[11]
//     Term 10 (APS4322-7000)/APS Outputs/PhiE 2Y0 <-> Data Pointer/PhiSetPoints[15]
//     Term 10 (APS4322-7000)/APS Outputs/PhiE 2Y1 <-> Data Pointer/PhiSetPoints[16]
//     Term 10 (APS4322-7000)/APS Outputs/PhiE 2Y2 <-> Data Pointer/PhiSetPoints[17]
//     Term 10 (APS4322-7000)/APS Outputs/PhiE 3Y0 <-> Data Pointer/PhiSetPoints[21]
//     Term 10 (APS4322-7000)/APS Outputs/PhiE 3Y1 <-> Data Pointer/PhiSetPoints[22]
//     Term 10 (APS4322-7000)/APS Outputs/PhiE 3Y2 <-> Data Pointer/PhiSetPoints[23]
//     Term 10 (APS4322-7000)/Term 11 (APS4322-5000)/FB Inputs/A{0..8 step 2} X-Field <-> Data Pointer/HallSensorFieldsXYZ[{0..12 step 3}]  (5 links)
//     Term 10 (APS4322-7000)/Term 11 (APS4322-5000)/FB Inputs/A{0..8 step 2} Y-Field <-> Data Pointer/HallSensorFieldsXYZ[{1..13 step 3}]  (5 links)
//     Term 10 (APS4322-7000)/Term 11 (APS4322-5000)/FB Inputs/A{0..8 step 2} Z-Field <-> Data Pointer/HallSensorFieldsXYZ[{2..14 step 3}]  (5 links)
//     Term 10 (APS4322-7000)/Term 11 (APS4322-5000)/FB Inputs/B{1..9 step 2} X-Field <-> Data Pointer/HallSensorFieldsXYZ[{15..27 step 3}]  (5 links)
//     Term 10 (APS4322-7000)/Term 11 (APS4322-5000)/FB Inputs/B{1..9 step 2} Y-Field <-> Data Pointer/HallSensorFieldsXYZ[{16..28 step 3}]  (5 links)
//     Term 10 (APS4322-7000)/Term 11 (APS4322-5000)/FB Inputs/B{1..9 step 2} Z-Field <-> Data Pointer/HallSensorFieldsXYZ[{17..29 step 3}]  (5 links)
//     Term 10 (APS4322-7000)/Term 11 (APS4322-5000)/FB Inputs/C{0..8 step 2} X-Field <-> Data Pointer/HallSensorFieldsXYZ[{30..42 step 3}]  (5 links)
//     Term 10 (APS4322-7000)/Term 11 (APS4322-5000)/FB Inputs/C{0..8 step 2} Y-Field <-> Data Pointer/HallSensorFieldsXYZ[{31..43 step 3}]  (5 links)
//     Term 10 (APS4322-7000)/Term 11 (APS4322-5000)/FB Inputs/C{0..8 step 2} Z-Field <-> Data Pointer/HallSensorFieldsXYZ[{32..44 step 3}]  (5 links)
//     Term 10 (APS4322-7000)/Term 11 (APS4322-5000)/FB Inputs/D{1..9 step 2} X-Field <-> Data Pointer/HallSensorFieldsXYZ[{45..57 step 3}]  (5 links)
//     Term 10 (APS4322-7000)/Term 11 (APS4322-5000)/FB Inputs/D{1..9 step 2} Y-Field <-> Data Pointer/HallSensorFieldsXYZ[{46..58 step 3}]  (5 links)
//     Term 10 (APS4322-7000)/Term 11 (APS4322-5000)/FB Inputs/D{1..9 step 2} Z-Field <-> Data Pointer/HallSensorFieldsXYZ[{47..59 step 3}]  (5 links)
//     Term 10 (APS4322-7000)/Term 11 (APS4322-5000)/FB Inputs/E{0..8 step 2} X-Field <-> Data Pointer/HallSensorFieldsXYZ[{60..72 step 3}]  (5 links)
//     Term 10 (APS4322-7000)/Term 11 (APS4322-5000)/FB Inputs/E{0..8 step 2} Y-Field <-> Data Pointer/HallSensorFieldsXYZ[{61..73 step 3}]  (5 links)
//     Term 10 (APS4322-7000)/Term 11 (APS4322-5000)/FB Inputs/E{0..8 step 2} Z-Field <-> Data Pointer/HallSensorFieldsXYZ[{62..74 step 3}]  (5 links)
//     Term 10 (APS4322-7000)/Term 11 (APS4322-5000)/FB Inputs/F{1..9 step 2} X-Field <-> Data Pointer/HallSensorFieldsXYZ[{75..87 step 3}]  (5 links)
//     Term 10 (APS4322-7000)/Term 11 (APS4322-5000)/FB Inputs/F{1..9 step 2} Y-Field <-> Data Pointer/HallSensorFieldsXYZ[{76..88 step 3}]  (5 links)
//     Term 10 (APS4322-7000)/Term 11 (APS4322-5000)/FB Inputs/F{1..9 step 2} Z-Field <-> Data Pointer/HallSensorFieldsXYZ[{77..89 step 3}]  (5 links)
//     Term 10 (APS4322-7000)/Term 11 (APS4322-5000)/FB Inputs/G{0..8 step 2} X-Field <-> Data Pointer/HallSensorFieldsXYZ[{90..102 step 3}]  (5 links)
//     Term 10 (APS4322-7000)/Term 11 (APS4322-5000)/FB Inputs/G{0..8 step 2} Y-Field <-> Data Pointer/HallSensorFieldsXYZ[{91..103 step 3}]  (5 links)
//     Term 10 (APS4322-7000)/Term 11 (APS4322-5000)/FB Inputs/G{0..8 step 2} Z-Field <-> Data Pointer/HallSensorFieldsXYZ[{92..104 step 3}]  (5 links)
//     Term 10 (APS4322-7000)/Term 11 (APS4322-5000)/FB Inputs/H{1..9 step 2} X-Field <-> Data Pointer/HallSensorFieldsXYZ[{105..117 step 3}]  (5 links)
//     Term 10 (APS4322-7000)/Term 11 (APS4322-5000)/FB Inputs/H{1..9 step 2} Y-Field <-> Data Pointer/HallSensorFieldsXYZ[{106..118 step 3}]  (5 links)
//     Term 10 (APS4322-7000)/Term 11 (APS4322-5000)/FB Inputs/H{1..9 step 2} Z-Field <-> Data Pointer/HallSensorFieldsXYZ[{107..119 step 3}]  (5 links)
//     Term 10 (APS4322-7000)/Term 11 (APS4322-5000)/FB Inputs/I{0..8 step 2} X-Field <-> Data Pointer/HallSensorFieldsXYZ[{120..132 step 3}]  (5 links)
//     Term 10 (APS4322-7000)/Term 11 (APS4322-5000)/FB Inputs/I{0..8 step 2} Y-Field <-> Data Pointer/HallSensorFieldsXYZ[{121..133 step 3}]  (5 links)
//     Term 10 (APS4322-7000)/Term 11 (APS4322-5000)/FB Inputs/I{0..8 step 2} Z-Field <-> Data Pointer/HallSensorFieldsXYZ[{122..134 step 3}]  (5 links)
//     Term 10 (APS4322-7000)/Term 11 (APS4322-5000)/FB Inputs/J{1..9 step 2} X-Field <-> Data Pointer/HallSensorFieldsXYZ[{135..147 step 3}]  (5 links)
//     Term 10 (APS4322-7000)/Term 11 (APS4322-5000)/FB Inputs/J{1..9 step 2} Y-Field <-> Data Pointer/HallSensorFieldsXYZ[{136..148 step 3}]  (5 links)
//     Term 10 (APS4322-7000)/Term 11 (APS4322-5000)/FB Inputs/J{1..9 step 2} Z-Field <-> Data Pointer/HallSensorFieldsXYZ[{137..149 step 3}]  (5 links)
//     Term 10 (APS4322-7000)/Term 11 (APS4322-5000)/FB Inputs/Status <-> Data Pointer/FeedbackStatus
//   Device 5 (EtherCAT) <-> TcCOM Objects/XPlanar/Part1/APS4322_P1_6
//     Term 8 (APS4322-7000)/APS Comm Inputs/CommStatusWord <-> Data Pointer/MoverCommStatusWord
//     Term 8 (APS4322-7000)/APS Comm Inputs/Data {1..4} <-> Data Pointer/MoverCommDataIn[{0..3}]  (4 links)
//     Term 8 (APS4322-7000)/APS Comm Outputs/CommControlWord <-> Data Pointer/MoverCommControlWord
//     Term 8 (APS4322-7000)/APS Comm Outputs/Data 1 <-> Data Pointer/MoverCommDataOut
//     Term 8 (APS4322-7000)/APS Diagdata/DC Link Voltage <-> Data Pointer/DcLinkVoltage
//     Term 8 (APS4322-7000)/APS Diagdata/Power supply current <-> Data Pointer/PowerSupplyCurrent
//     Term 8 (APS4322-7000)/APS Inputs/StatusWord <-> Data Pointer/PowerUnitStatusWord
//     Term 8 (APS4322-7000)/APS Outputs/ControlWord <-> Data Pointer/PowerUnitControlWord
//     Term 8 (APS4322-7000)/APS Outputs/Current D 0X0 <-> Data Pointer/DCurrentSetPoints[0]
//     Term 8 (APS4322-7000)/APS Outputs/Current D 0X1 <-> Data Pointer/DCurrentSetPoints[1]
//     Term 8 (APS4322-7000)/APS Outputs/Current D 0X2 <-> Data Pointer/DCurrentSetPoints[2]
//     Term 8 (APS4322-7000)/APS Outputs/Current D 1X0 <-> Data Pointer/DCurrentSetPoints[6]
//     Term 8 (APS4322-7000)/APS Outputs/Current D 1X1 <-> Data Pointer/DCurrentSetPoints[7]
//     Term 8 (APS4322-7000)/APS Outputs/Current D 1X2 <-> Data Pointer/DCurrentSetPoints[8]
//     Term 8 (APS4322-7000)/APS Outputs/Current D 2X0 <-> Data Pointer/DCurrentSetPoints[12]
//     Term 8 (APS4322-7000)/APS Outputs/Current D 2X1 <-> Data Pointer/DCurrentSetPoints[13]
//     Term 8 (APS4322-7000)/APS Outputs/Current D 2X2 <-> Data Pointer/DCurrentSetPoints[14]
//     Term 8 (APS4322-7000)/APS Outputs/Current D 3X0 <-> Data Pointer/DCurrentSetPoints[18]
//     Term 8 (APS4322-7000)/APS Outputs/Current D 3X1 <-> Data Pointer/DCurrentSetPoints[19]
//     Term 8 (APS4322-7000)/APS Outputs/Current D 3X2 <-> Data Pointer/DCurrentSetPoints[20]
//     Term 8 (APS4322-7000)/APS Outputs/Current D 0Y0 <-> Data Pointer/DCurrentSetPoints[3]
//     Term 8 (APS4322-7000)/APS Outputs/Current D 0Y1 <-> Data Pointer/DCurrentSetPoints[4]
//     Term 8 (APS4322-7000)/APS Outputs/Current D 0Y2 <-> Data Pointer/DCurrentSetPoints[5]
//     Term 8 (APS4322-7000)/APS Outputs/Current D 1Y0 <-> Data Pointer/DCurrentSetPoints[9]
//     Term 8 (APS4322-7000)/APS Outputs/Current D 1Y1 <-> Data Pointer/DCurrentSetPoints[10]
//     Term 8 (APS4322-7000)/APS Outputs/Current D 1Y2 <-> Data Pointer/DCurrentSetPoints[11]
//     Term 8 (APS4322-7000)/APS Outputs/Current D 2Y0 <-> Data Pointer/DCurrentSetPoints[15]
//     Term 8 (APS4322-7000)/APS Outputs/Current D 2Y1 <-> Data Pointer/DCurrentSetPoints[16]
//     Term 8 (APS4322-7000)/APS Outputs/Current D 2Y2 <-> Data Pointer/DCurrentSetPoints[17]
//     Term 8 (APS4322-7000)/APS Outputs/Current D 3Y0 <-> Data Pointer/DCurrentSetPoints[21]
//     Term 8 (APS4322-7000)/APS Outputs/Current D 3Y1 <-> Data Pointer/DCurrentSetPoints[22]
//     Term 8 (APS4322-7000)/APS Outputs/Current D 3Y2 <-> Data Pointer/DCurrentSetPoints[23]
//     Term 8 (APS4322-7000)/APS Outputs/Current Q 0X0 <-> Data Pointer/QCurrentSetPoints[0]
//     Term 8 (APS4322-7000)/APS Outputs/Current Q 0X1 <-> Data Pointer/QCurrentSetPoints[1]
//     Term 8 (APS4322-7000)/APS Outputs/Current Q 0X2 <-> Data Pointer/QCurrentSetPoints[2]
//     Term 8 (APS4322-7000)/APS Outputs/Current Q 1X0 <-> Data Pointer/QCurrentSetPoints[6]
//     Term 8 (APS4322-7000)/APS Outputs/Current Q 1X1 <-> Data Pointer/QCurrentSetPoints[7]
//     Term 8 (APS4322-7000)/APS Outputs/Current Q 1X2 <-> Data Pointer/QCurrentSetPoints[8]
//     Term 8 (APS4322-7000)/APS Outputs/Current Q 2X0 <-> Data Pointer/QCurrentSetPoints[12]
//     Term 8 (APS4322-7000)/APS Outputs/Current Q 2X1 <-> Data Pointer/QCurrentSetPoints[13]
//     Term 8 (APS4322-7000)/APS Outputs/Current Q 2X2 <-> Data Pointer/QCurrentSetPoints[14]
//     Term 8 (APS4322-7000)/APS Outputs/Current Q 3X0 <-> Data Pointer/QCurrentSetPoints[18]
//     Term 8 (APS4322-7000)/APS Outputs/Current Q 3X1 <-> Data Pointer/QCurrentSetPoints[19]
//     Term 8 (APS4322-7000)/APS Outputs/Current Q 3X2 <-> Data Pointer/QCurrentSetPoints[20]
//     Term 8 (APS4322-7000)/APS Outputs/Current Q 0Y0 <-> Data Pointer/QCurrentSetPoints[3]
//     Term 8 (APS4322-7000)/APS Outputs/Current Q 0Y1 <-> Data Pointer/QCurrentSetPoints[4]
//     Term 8 (APS4322-7000)/APS Outputs/Current Q 0Y2 <-> Data Pointer/QCurrentSetPoints[5]
//     Term 8 (APS4322-7000)/APS Outputs/Current Q 1Y0 <-> Data Pointer/QCurrentSetPoints[9]
//     Term 8 (APS4322-7000)/APS Outputs/Current Q 1Y1 <-> Data Pointer/QCurrentSetPoints[10]
//     Term 8 (APS4322-7000)/APS Outputs/Current Q 1Y2 <-> Data Pointer/QCurrentSetPoints[11]
//     Term 8 (APS4322-7000)/APS Outputs/Current Q 2Y0 <-> Data Pointer/QCurrentSetPoints[15]
//     Term 8 (APS4322-7000)/APS Outputs/Current Q 2Y1 <-> Data Pointer/QCurrentSetPoints[16]
//     Term 8 (APS4322-7000)/APS Outputs/Current Q 2Y2 <-> Data Pointer/QCurrentSetPoints[17]
//     Term 8 (APS4322-7000)/APS Outputs/Current Q 3Y0 <-> Data Pointer/QCurrentSetPoints[21]
//     Term 8 (APS4322-7000)/APS Outputs/Current Q 3Y1 <-> Data Pointer/QCurrentSetPoints[22]
//     Term 8 (APS4322-7000)/APS Outputs/Current Q 3Y2 <-> Data Pointer/QCurrentSetPoints[23]
//     Term 8 (APS4322-7000)/APS Outputs/PhiE 0X0 <-> Data Pointer/PhiSetPoints[0]
//     Term 8 (APS4322-7000)/APS Outputs/PhiE 0X1 <-> Data Pointer/PhiSetPoints[1]
//     Term 8 (APS4322-7000)/APS Outputs/PhiE 0X2 <-> Data Pointer/PhiSetPoints[2]
//     Term 8 (APS4322-7000)/APS Outputs/PhiE 1X0 <-> Data Pointer/PhiSetPoints[6]
//     Term 8 (APS4322-7000)/APS Outputs/PhiE 1X1 <-> Data Pointer/PhiSetPoints[7]
//     Term 8 (APS4322-7000)/APS Outputs/PhiE 1X2 <-> Data Pointer/PhiSetPoints[8]
//     Term 8 (APS4322-7000)/APS Outputs/PhiE 2X0 <-> Data Pointer/PhiSetPoints[12]
//     Term 8 (APS4322-7000)/APS Outputs/PhiE 2X1 <-> Data Pointer/PhiSetPoints[13]
//     Term 8 (APS4322-7000)/APS Outputs/PhiE 2X2 <-> Data Pointer/PhiSetPoints[14]
//     Term 8 (APS4322-7000)/APS Outputs/PhiE 3X0 <-> Data Pointer/PhiSetPoints[18]
//     Term 8 (APS4322-7000)/APS Outputs/PhiE 3X1 <-> Data Pointer/PhiSetPoints[19]
//     Term 8 (APS4322-7000)/APS Outputs/PhiE 3X2 <-> Data Pointer/PhiSetPoints[20]
//     Term 8 (APS4322-7000)/APS Outputs/PhiE 0Y0 <-> Data Pointer/PhiSetPoints[3]
//     Term 8 (APS4322-7000)/APS Outputs/PhiE 0Y1 <-> Data Pointer/PhiSetPoints[4]
//     Term 8 (APS4322-7000)/APS Outputs/PhiE 0Y2 <-> Data Pointer/PhiSetPoints[5]
//     Term 8 (APS4322-7000)/APS Outputs/PhiE 1Y0 <-> Data Pointer/PhiSetPoints[9]
//     Term 8 (APS4322-7000)/APS Outputs/PhiE 1Y1 <-> Data Pointer/PhiSetPoints[10]
//     Term 8 (APS4322-7000)/APS Outputs/PhiE 1Y2 <-> Data Pointer/PhiSetPoints[11]
//     Term 8 (APS4322-7000)/APS Outputs/PhiE 2Y0 <-> Data Pointer/PhiSetPoints[15]
//     Term 8 (APS4322-7000)/APS Outputs/PhiE 2Y1 <-> Data Pointer/PhiSetPoints[16]
//     Term 8 (APS4322-7000)/APS Outputs/PhiE 2Y2 <-> Data Pointer/PhiSetPoints[17]
//     Term 8 (APS4322-7000)/APS Outputs/PhiE 3Y0 <-> Data Pointer/PhiSetPoints[21]
//     Term 8 (APS4322-7000)/APS Outputs/PhiE 3Y1 <-> Data Pointer/PhiSetPoints[22]
//     Term 8 (APS4322-7000)/APS Outputs/PhiE 3Y2 <-> Data Pointer/PhiSetPoints[23]
//     Term 8 (APS4322-7000)/Term 9 (APS4322-5000)/FB Inputs/A{0..8 step 2} X-Field <-> Data Pointer/HallSensorFieldsXYZ[{0..12 step 3}]  (5 links)
//     Term 8 (APS4322-7000)/Term 9 (APS4322-5000)/FB Inputs/A{0..8 step 2} Y-Field <-> Data Pointer/HallSensorFieldsXYZ[{1..13 step 3}]  (5 links)
//     Term 8 (APS4322-7000)/Term 9 (APS4322-5000)/FB Inputs/A{0..8 step 2} Z-Field <-> Data Pointer/HallSensorFieldsXYZ[{2..14 step 3}]  (5 links)
//     Term 8 (APS4322-7000)/Term 9 (APS4322-5000)/FB Inputs/B{1..9 step 2} X-Field <-> Data Pointer/HallSensorFieldsXYZ[{15..27 step 3}]  (5 links)
//     Term 8 (APS4322-7000)/Term 9 (APS4322-5000)/FB Inputs/B{1..9 step 2} Y-Field <-> Data Pointer/HallSensorFieldsXYZ[{16..28 step 3}]  (5 links)
//     Term 8 (APS4322-7000)/Term 9 (APS4322-5000)/FB Inputs/B{1..9 step 2} Z-Field <-> Data Pointer/HallSensorFieldsXYZ[{17..29 step 3}]  (5 links)
//     Term 8 (APS4322-7000)/Term 9 (APS4322-5000)/FB Inputs/C{0..8 step 2} X-Field <-> Data Pointer/HallSensorFieldsXYZ[{30..42 step 3}]  (5 links)
//     Term 8 (APS4322-7000)/Term 9 (APS4322-5000)/FB Inputs/C{0..8 step 2} Y-Field <-> Data Pointer/HallSensorFieldsXYZ[{31..43 step 3}]  (5 links)
//     Term 8 (APS4322-7000)/Term 9 (APS4322-5000)/FB Inputs/C{0..8 step 2} Z-Field <-> Data Pointer/HallSensorFieldsXYZ[{32..44 step 3}]  (5 links)
//     Term 8 (APS4322-7000)/Term 9 (APS4322-5000)/FB Inputs/D{1..9 step 2} X-Field <-> Data Pointer/HallSensorFieldsXYZ[{45..57 step 3}]  (5 links)
//     Term 8 (APS4322-7000)/Term 9 (APS4322-5000)/FB Inputs/D{1..9 step 2} Y-Field <-> Data Pointer/HallSensorFieldsXYZ[{46..58 step 3}]  (5 links)
//     Term 8 (APS4322-7000)/Term 9 (APS4322-5000)/FB Inputs/D{1..9 step 2} Z-Field <-> Data Pointer/HallSensorFieldsXYZ[{47..59 step 3}]  (5 links)
//     Term 8 (APS4322-7000)/Term 9 (APS4322-5000)/FB Inputs/E{0..8 step 2} X-Field <-> Data Pointer/HallSensorFieldsXYZ[{60..72 step 3}]  (5 links)
//     Term 8 (APS4322-7000)/Term 9 (APS4322-5000)/FB Inputs/E{0..8 step 2} Y-Field <-> Data Pointer/HallSensorFieldsXYZ[{61..73 step 3}]  (5 links)
//     Term 8 (APS4322-7000)/Term 9 (APS4322-5000)/FB Inputs/E{0..8 step 2} Z-Field <-> Data Pointer/HallSensorFieldsXYZ[{62..74 step 3}]  (5 links)
//     Term 8 (APS4322-7000)/Term 9 (APS4322-5000)/FB Inputs/F{1..9 step 2} X-Field <-> Data Pointer/HallSensorFieldsXYZ[{75..87 step 3}]  (5 links)
//     Term 8 (APS4322-7000)/Term 9 (APS4322-5000)/FB Inputs/F{1..9 step 2} Y-Field <-> Data Pointer/HallSensorFieldsXYZ[{76..88 step 3}]  (5 links)
//     Term 8 (APS4322-7000)/Term 9 (APS4322-5000)/FB Inputs/F{1..9 step 2} Z-Field <-> Data Pointer/HallSensorFieldsXYZ[{77..89 step 3}]  (5 links)
//     Term 8 (APS4322-7000)/Term 9 (APS4322-5000)/FB Inputs/G{0..8 step 2} X-Field <-> Data Pointer/HallSensorFieldsXYZ[{90..102 step 3}]  (5 links)
//     Term 8 (APS4322-7000)/Term 9 (APS4322-5000)/FB Inputs/G{0..8 step 2} Y-Field <-> Data Pointer/HallSensorFieldsXYZ[{91..103 step 3}]  (5 links)
//     Term 8 (APS4322-7000)/Term 9 (APS4322-5000)/FB Inputs/G{0..8 step 2} Z-Field <-> Data Pointer/HallSensorFieldsXYZ[{92..104 step 3}]  (5 links)
//     Term 8 (APS4322-7000)/Term 9 (APS4322-5000)/FB Inputs/H{1..9 step 2} X-Field <-> Data Pointer/HallSensorFieldsXYZ[{105..117 step 3}]  (5 links)
//     Term 8 (APS4322-7000)/Term 9 (APS4322-5000)/FB Inputs/H{1..9 step 2} Y-Field <-> Data Pointer/HallSensorFieldsXYZ[{106..118 step 3}]  (5 links)
//     Term 8 (APS4322-7000)/Term 9 (APS4322-5000)/FB Inputs/H{1..9 step 2} Z-Field <-> Data Pointer/HallSensorFieldsXYZ[{107..119 step 3}]  (5 links)
//     Term 8 (APS4322-7000)/Term 9 (APS4322-5000)/FB Inputs/I{0..8 step 2} X-Field <-> Data Pointer/HallSensorFieldsXYZ[{120..132 step 3}]  (5 links)
//     Term 8 (APS4322-7000)/Term 9 (APS4322-5000)/FB Inputs/I{0..8 step 2} Y-Field <-> Data Pointer/HallSensorFieldsXYZ[{121..133 step 3}]  (5 links)
//     Term 8 (APS4322-7000)/Term 9 (APS4322-5000)/FB Inputs/I{0..8 step 2} Z-Field <-> Data Pointer/HallSensorFieldsXYZ[{122..134 step 3}]  (5 links)
//     Term 8 (APS4322-7000)/Term 9 (APS4322-5000)/FB Inputs/J{1..9 step 2} X-Field <-> Data Pointer/HallSensorFieldsXYZ[{135..147 step 3}]  (5 links)
//     Term 8 (APS4322-7000)/Term 9 (APS4322-5000)/FB Inputs/J{1..9 step 2} Y-Field <-> Data Pointer/HallSensorFieldsXYZ[{136..148 step 3}]  (5 links)
//     Term 8 (APS4322-7000)/Term 9 (APS4322-5000)/FB Inputs/J{1..9 step 2} Z-Field <-> Data Pointer/HallSensorFieldsXYZ[{137..149 step 3}]  (5 links)
//     Term 8 (APS4322-7000)/Term 9 (APS4322-5000)/FB Inputs/Status <-> Data Pointer/FeedbackStatus
//   XPlanar MC Project/Axes/Mover4220_1 <-> TcCOM Objects/XPlanar/Mover4220_1
//     IoToMc/STD <-> OutputsToNC3/HWToNC3
//     McToIo/STD <-> InputsFromNC3/NC3ToHW
//   XPlanar MC Project/Axes/Mover4220_2 <-> TcCOM Objects/XPlanar/Mover4220_2
//     IoToMc/STD <-> OutputsToNC3/HWToNC3
//     McToIo/STD <-> InputsFromNC3/NC3ToHW
//   XPlanar MC Project/Axes/Mover4220_3 <-> TcCOM Objects/XPlanar/Mover4220_3
//     IoToMc/STD <-> OutputsToNC3/HWToNC3
//     McToIo/STD <-> InputsFromNC3/NC3ToHW
//   XPlanar MC Project/Axes/Mover4220_4 <-> TcCOM Objects/XPlanar/Mover4220_4
//     IoToMc/STD <-> OutputsToNC3/HWToNC3
//     McToIo/STD <-> InputsFromNC3/NC3ToHW
//   Test_PLC/Test_PLC Instance <-> Device 1 (TC3 EIP Adapter)/Box 20 (TC EtherNet/IP Slave)
//     PlcTask Inputs/MAIN.iEipInput <-> Assembly 1 (Input/Output)/Inputs/AssemblyEIPinput
//   Test_PLC/Test_PLC Instance <-> Device 4 (EtherCAT)/Term 1 (EK1100)/Term 2 (EL1008)
//     PlcTask Inputs/GVL.inputl <-> Channel 1/Input
//     PlcTask Inputs/MAIN.bSlowStop <-> Channel 7/Input
//   Test_PLC/Test_PLC Instance <-> Device 4 (EtherCAT)/Term 1 (EK1100)/Term 3 (EL2008-0015)
//     PlcTask Outputs/GVL.output2 <-> Channel 1/Output
//   Test_PLC/Test_PLC Instance <-> XPlanar MC Project/Axes/Mover4220_1
//     PlcTask Inputs/MAIN.Xpmover[0].MCTOPLC/ACT <-> McToPlc/ACT
//     PlcTask Inputs/MAIN.Xpmover[0].MCTOPLC/COORDMODE <-> McToPlc/COORDMODE
//     PlcTask Inputs/MAIN.Xpmover[0].MCTOPLC/SET <-> McToPlc/SET
//     PlcTask Inputs/MAIN.Xpmover[0].MCTOPLC/SETONTRACK <-> McToPlc/SETONTRACK
//     PlcTask Inputs/MAIN.Xpmover[0].MCTOPLC/STD <-> McToPlc/STD
//     PlcTask Outputs/MAIN.Xpmover[0].PLCTOMC/STD <-> PlcToMc/STD
//   Test_PLC/Test_PLC Instance <-> XPlanar MC Project/Axes/Mover4220_2
//     PlcTask Inputs/MAIN.Xpmover[1].MCTOPLC/ACT <-> McToPlc/ACT
//     PlcTask Inputs/MAIN.Xpmover[1].MCTOPLC/COORDMODE <-> McToPlc/COORDMODE
//     PlcTask Inputs/MAIN.Xpmover[1].MCTOPLC/SET <-> McToPlc/SET
//     PlcTask Inputs/MAIN.Xpmover[1].MCTOPLC/SETONTRACK <-> McToPlc/SETONTRACK
//     PlcTask Inputs/MAIN.Xpmover[1].MCTOPLC/STD <-> McToPlc/STD
//     PlcTask Outputs/MAIN.Xpmover[1].PLCTOMC/STD <-> PlcToMc/STD
//   Test_PLC/Test_PLC Instance <-> XPlanar MC Project/Axes/Mover4220_3
//     PlcTask Inputs/MAIN.Xpmover[2].MCTOPLC/ACT <-> McToPlc/ACT
//     PlcTask Inputs/MAIN.Xpmover[2].MCTOPLC/COORDMODE <-> McToPlc/COORDMODE
//     PlcTask Inputs/MAIN.Xpmover[2].MCTOPLC/SET <-> McToPlc/SET
//     PlcTask Inputs/MAIN.Xpmover[2].MCTOPLC/SETONTRACK <-> McToPlc/SETONTRACK
//     PlcTask Inputs/MAIN.Xpmover[2].MCTOPLC/STD <-> McToPlc/STD
//     PlcTask Outputs/MAIN.Xpmover[2].PLCTOMC/STD <-> PlcToMc/STD
//   Test_PLC/Test_PLC Instance <-> XPlanar MC Project/Axes/Mover4220_4
//     PlcTask Inputs/MAIN.Xpmover[3].MCTOPLC/ACT <-> McToPlc/ACT
//     PlcTask Inputs/MAIN.Xpmover[3].MCTOPLC/COORDMODE <-> McToPlc/COORDMODE
//     PlcTask Inputs/MAIN.Xpmover[3].MCTOPLC/SET <-> McToPlc/SET
//     PlcTask Inputs/MAIN.Xpmover[3].MCTOPLC/SETONTRACK <-> McToPlc/SETONTRACK
//     PlcTask Inputs/MAIN.Xpmover[3].MCTOPLC/STD <-> McToPlc/STD
//     PlcTask Outputs/MAIN.Xpmover[3].PLCTOMC/STD <-> PlcToMc/STD
//   Test_PLC/Test_PLC Instance <-> XPlanar MC Project/Groups/EndA
//     PlcTask Inputs/MAIN.XpTrack[5].MCTOPLC_STD <-> McToPlc/STD
//   Test_PLC/Test_PLC Instance <-> XPlanar MC Project/Groups/EndB
//     PlcTask Inputs/MAIN.XpTrack[6].MCTOPLC_STD <-> McToPlc/STD
//   Test_PLC/Test_PLC Instance <-> XPlanar MC Project/Groups/ToCapA
//     PlcTask Inputs/MAIN.XpTrack[4].MCTOPLC_STD <-> McToPlc/STD
//   Test_PLC/Test_PLC Instance <-> XPlanar MC Project/Groups/ToCapB
//     PlcTask Inputs/MAIN.XpTrack[3].MCTOPLC_STD <-> McToPlc/STD
//   Test_PLC/Test_PLC Instance <-> XPlanar MC Project/Groups/ToFillA
//     PlcTask Inputs/MAIN.XpTrack[2].MCTOPLC_STD <-> McToPlc/STD
//   Test_PLC/Test_PLC Instance <-> XPlanar MC Project/Groups/ToFillB
//     PlcTask Inputs/MAIN.XpTrack[1].MCTOPLC_STD <-> McToPlc/STD
//   Test_PLC/Test_PLC Instance <-> XPlanar MC Project/Groups/Wait
//     PlcTask Inputs/MAIN.XpTrack[0].MCTOPLC_STD <-> McToPlc/STD

// ---- DUTs/ST_MoverFeedback.TcDUT
TYPE ST_MoverFeedback :
STRUCT
	CallEnable			: MC_PlanarFeedback;
	CallDisable			: MC_PlanarFeedback;
	CallHalt			: MC_PlanarFeedback;
	CallJoinTrack		: MC_PlanarFeedback;
	CallLeaveTrack		: MC_PlanarFeedback;
	CallReset			: MC_PlanarFeedback;
	CallMoveX			: MC_PlanarFeedback;
	CallMoveY			: MC_PlanarFeedback;
	CallMoveZ			: MC_PlanarFeedback;
	CallMoveA			: MC_PlanarFeedback;
	CallMoveB			: MC_PlanarFeedback;
	CallMoveC			: MC_PlanarFeedback;
	CallMoveOnTrack		: MC_PlanarFeedback;
	CallEmergencyStop	: MC_PlanarFeedback;
	SeqJoinTrack		: MC_PlanarFeedback;
	
END_STRUCT
END_TYPE
//Feedback変数を構造体にして、Feedbackの名称を明示

// ---- DUTs/U_MoverFeedback.TcDUT
TYPE U_MoverFeedback :
UNION
	sName	:ST_MoverFeedback;
	aArray	:ARRAY[0..GVL.MAX_FEEDBACK] OF MC_PlanarFeedback;
END_UNION
END_TYPE
//構造体で記載したFeedbackをUpdateする時にFORで処理できるように、同じ要素数の配列と同期する。

// ---- GVLs/GVL.TcGVL
{attribute 'qualified_only'}
VAR_GLOBAL
	inputl   AT%I*   :BOOL;
	output2  AT%Q*  :BOOL;
	JoinTrack: INT;
	
	bBusyA:BOOL;
	bBusyB:BOOL;
	bDoneA:BOOL;
	bDoneB:BOOL;
	bfill:BOOL;
	bstop:BOOL;

END_VAR

VAR_GLOBAL CONSTANT
	MAX_MOVER     :INT:=3; //0 to...
	MAX_FEEDBACK  :INT:=100;
	MAX_Track     :INT:=7;
END_VAR

// ---- POUs/FB_StateTrackMove.TcPOU
FUNCTION_BLOCK FB_StateTrackMove
VAR_IN_OUT
	Fbmover          :MC_PlanarMover;
	FbTrack          :ARRAY [*]OF MC_PlanarTrack;
END_VAR
VAR_INPUT
	bMoveState		: BOOL;
	bstart:BOOL;
	breset: BOOL;
	bEmergencyStopIn: BOOL;
END_VAR
VAR_OUTPUT
	icount: INT;
END_VAR
VAR
	Fbfeedback       :ARRAY [0..10]OF MC_Planarfeedback;
	iStateTrack		: INT;
	constraint_xy	: DynamicConstraint_PathXY;
	constraint_c	: DynamicConstraint_Coordinates;
	
	ValuePara		: ARRAY [0..5] OF INT;
	
	Value: INT:=200;
	Acc: INT:=3000;
	Dec: INT:=3000;
	Jerk: INT:=30000;
	
	TWait:ARRAY [0..5]OF  TON;
	
	xpm: LREAL;
	i: INT;
	bTimer: ARRAY [0..3]OF BOOL;
	bGoAline : BOOL;
	TrackName : E_TrackName;
	ValueC : INT:=600;
	bfillin : BOOL;
	bstop: BOOL;
	iCurrentState: INT;
END_VAR

IF bstart THEN
	iStateTrack:=0;
	bGoAline:=FALSE;
	
END_IF

IF breset THEN
	bReset := FALSE;
		icount:=0;
END_IF

IF NOT bEmergencyStopIn THEN
	iStateTrack := 999;
END_IF

CASE iStateTrack OF
	0://init and ready
	IF bMoveState THEN
		bMoveState := FALSE;
		iStateTrack :=10;
	END_IF
	
	10://move wait pos.
	Value :=100;
	TrackName:= E_TrackName.wait;
	Fbmover.MoveOnTrack(
	commandFeedback:= Fbfeedback[0], 
	targetTrack:= fbTrack[TrackName], 
	targetPositionOnTrack:= FbTrack[TrackName].GetLength(), 
	constraint:= constraint_xy, 
	options:= 0);
	iStateTrack:= 11;
	
	11:
	IF Fbfeedback[0].Done THEN
		iStateTrack :=19;
	END_IF
	
	19:
	Value :=200;
	iStateTrack :=20;
	
	20:
	//Value :=200;
	IF NOT gvl.bBusyA THEN
		bGoAline:=TRUE;
		TrackName := E_trackName.ToFillA;
		gvl.bBusyA:= TRUE;
	ELSE
		TrackName := E_trackname.ToFillB;
		gvl.bBusyB:= TRUE;
	END_IF
	Fbmover.MoveOnTrack(
	commandFeedback:= Fbfeedback[1], 
	targetTrack:= fbTrack[TrackName], 
	targetPositionOnTrack:= FbTrack[TrackName].GetLength(), 
	constraint:= constraint_xy, 
	options:= 0);
	iStateTrack:= 21;
	
	21:
	//IF Fbfeedback[1].Done THEN
	IF (gvl.bBusyA AND gvl.bBusyB)THEN;
		bTimer[0]:=TRUE;
		IF TWait[0].Q THEN
			bTimer[0]:=FALSE;
			iStateTrack:=29;
		END_IF
		(*IF gvl.bfill THEN
			iStateTrack:=29;
		END_IF*)
	END_IF
	
	29:
	Value :=200;
	iStateTrack :=30;
	
	30:
	//Value :=200;
	IF bGoAline THEN
		//bGoAline := FALSE;
		TrackName := E_trackName.TocapA;
		GVL.bBusyA:= FALSE;
	ELSE
		TrackName := E_trackname.ToCapB;
		GVL.bBusyB:= FALSE;
	END_IF
	IF  (NOT gvl.bDoneA AND NOT gvl.bDoneB) THEN 
	Fbmover.MoveOnTrack(
	commandFeedback:= Fbfeedback[2], 
	targetTrack:= fbTrack[TrackName], 
	targetPositionOnTrack:= FbTrack[TrackName].GetLength(), 
	constraint:= constraint_xy, 
	options:= 0);
	iStateTrack:= 31;
	END_IF

	31:
	IF Fbfeedback[2].Done THEN
		IF bGoAline THEN 
			gvl.bDoneA :=TRUE;
		ELSE
			gvl.bDoneB :=TRUE;
		END_IF
		IF (gvl.bDoneA AND gvl.bDoneB) THEN;
			bTimer[1]:=TRUE;
			IF TWait[1].Q THEN
				bTimer[1]:=FALSE;
				iStateTrack:=32;
			END_IF
		END_IF
	END_IF	
	
	
	
	32:
	//Value :=600;
	Fbmover.MoveC(commandFeedback:= Fbfeedback[3], 
	targetPosition:= fbmover.MCTOPLC.set.SetPos.c+720 , 
	constraint:= constraint_c,
	options:=0 );
	iStateTrack:= 33;
	
	33:
	IF Fbfeedback[3].Done THEN
		bTimer[2]:=TRUE;
		IF TWait[2].Q THEN
			bTimer[2]:=FALSE;
			iStateTrack:=39;
		END_IF
	END_IF	
	
	39:
	Value :=400;
	iStateTrack :=40;
	
	40:
	//Value :=1000;
	bGoAline := FALSE;
	GVL.bDoneA:= FALSE;
	GVL.bDoneB:= FALSE;
	TrackName:= E_TrackName.Wait;
	Fbmover.MoveOnTrack(
	commandFeedback:= Fbfeedback[4], 
	targetTrack:= fbTrack[TrackName], 
	targetPositionOnTrack:= FbTrack[TrackName].GetLength(), 
	constraint:= constraint_xy, 
	options:= 0);
	IF gvl.bstop THEN
		iStatetrack := 19;
	END_IF
	iStateTrack:= 41;
	
	41:
		icount:=icount+1;
		iStateTrack := 42;
		
	42:
	IF gvl.bstop THEN
		iCurrentState := iStateTrack;
		iStateTrack := 100;
	END_IF	
	IF Fbfeedback[4].Done AND NOT gvl.bstop THEN
		iStateTrack:=19;	
	END_IF
	
	100:
	IF NOT gvl.bstop THEN
		iStateTrack := iCurrentState;
	END_IF
	
	999:
	IF bEmergencyStopIn THEN
		iStateTrack := 0;
	END_IF
	
	
END_CASE

constraint_xy.SetValuesVADJ(v:=Value,A:=Acc,D:=Dec,j:=Jerk);
constraint_c.SetLimit(Coordinate:=Coord_Mcs_C1,v:=ValueC,A:=Acc,D:=Dec,j:=Jerk);

TWait[0](IN:=bTimer[0],PT:=T#4S);
TWait[1](IN:=bTimer[1],PT:=T#1S);
TWait[2](IN:=bTimer[2],PT:=T#2S);

FOR i:=0 TO 10 DO
	Fbfeedback[i].Update();
END_FOR

END_FUNCTION_BLOCK

// ---- POUs/MAIN.TcPOU
PROGRAM MAIN
VAR
	seqEnableM       :ARRAY[0..gvl.MAX_mover]OF UINT;
	enableM          :ARRAY[0..gvl.MAX_mover]OF BOOL;
	ResetM           :ARRAY[0..gvl.MAX_mover]OF BOOL;
	seqResetM        :ARRAY[0..gvl.MAX_mover]OF UINT;
	HaltM            :ARRAY[0..gvl.MAX_mover]OF BOOL;
	seqHaltM         :ARRAY[0..gvl.MAX_mover]OF UINT;
	seqdisableM      :ARRAY[0..gvl.MAX_mover]OF UINT;
	disableM         :ARRAY[0..gvl.MAX_mover]OF BOOL;
	seqMovexM        :ARRAY[0..gvl.MAX_mover]OF UINT;
	seqMoveX_2m      :UINT;
	seqMoveAM        :ARRAY[0..gvl.MAX_mover]OF UINT;
	seqMovex1M       :ARRAY[0..gvl.MAX_mover]OF UINT;
	moveXM           :ARRAY[0..gvl.MAX_mover]OF BOOL;
	moveAM           :ARRAY[0..gvl.MAX_mover]OF BOOL;
	moveX1M          :ARRAY[0..gvl.MAX_mover]OF BOOL;
	MoveX_2m         :BOOL;
	moveZM           :ARRAY[0..gvl.MAX_mover]OF BOOL;
	moveCM           :ARRAY[0..gvl.MAX_mover]OF BOOL;
	positionTargetX  :ARRAY[0..gvl.MAX_mover]OF LREAL :=[(gvl.MAX_MOVER+1)(120)];
	positionTargetA  :ARRAY[0..gvl.MAX_mover]OF LREAL :=[(gvl.MAX_MOVER+1)(0)];
	positionTargetX1 :ARRAY[0..gvl.MAX_mover]OF LREAL :=[(gvl.MAX_MOVER+1)(140)];
	seqMoveYM        :ARRAY[0..gvl.MAX_mover]OF UINT;
	seqMoveBM        :ARRAY[0..gvl.MAX_mover]OF UINT;
	seqMoveCM        :ARRAY[0..gvl.MAX_mover]OF UINT;
	seqMoveZM        :ARRAY[0..gvl.MAX_mover]OF UINT;
	seqMoveY1M       :ARRAY[0..gvl.MAX_mover]OF UINT;
	seqJoinTrack     :ARRAY[0..gvl.MAX_mover]OF UINT;
	seqLeaveTrack    :ARRAY[0..gvl.MAX_mover]OF UINT;
	seqMoveOnTrack   :ARRAY[0..gvl.MAX_mover]OF UINT;
	
	JoinTrack        :ARRAY[0..gvl.MAX_mover]OF BOOL;
	LeaveTrack       :ARRAY[0..gvl.MAX_mover]OF BOOL;
	MoveOnTrack      :ARRAY[0..gvl.MAX_mover]OF BOOL;
	moveYM           :ARRAY[0..gvl.MAX_mover]OF BOOL;
	moveBM           :ARRAY[0..gvl.MAX_mover]OF BOOL;
	moveY1M          :ARRAY[0..gvl.MAX_mover]OF BOOL;
	positionTargetY  :ARRAY[0..gvl.MAX_mover]OF LREAL :=[(gvl.MAX_MOVER+1)(120)];
	positionTargetB  :ARRAY[0..gvl.MAX_mover]OF LREAL :=[(gvl.MAX_MOVER+1)(0)];
	positionTargetC  :ARRAY[0..gvl.MAX_mover]OF LREAL :=[(gvl.MAX_MOVER+1)(0)];
	positionTargetZ  :ARRAY[0..gvl.MAX_mover]OF LREAL :=[(gvl.MAX_MOVER+1)(5)];
	positionTargetY1 :ARRAY[0..gvl.MAX_mover]OF LREAL :=[(gvl.MAX_MOVER+1)(140)];
	velocity_xy      :ARRAY[0..gvl.MAX_mover]OF LREAL :=[(gvl.MAX_MOVER+1)(50)];
	velocity_c       :ARRAY[0..gvl.MAX_mover]OF LREAL :=[(gvl.MAX_MOVER+1)(500)];
	velocity_ZAB     :ARRAY[0..gvl.MAX_mover]OF LREAL :=[(gvl.MAX_MOVER+1)(10)];
	Acc_xy     		 :ARRAY[0..gvl.MAX_mover]OF LREAL :=[(gvl.MAX_MOVER+1)(1000)];
	Jark_xy    		 :ARRAY[0..gvl.MAX_mover]OF LREAL :=[(gvl.MAX_MOVER+1)(1000)];
	PositionXYC      :ARRAY[0..gvl.MAX_mover]OF PositionXYC;
	numberTrack      :ARRAY[0..gvl.MAX_mover]OF  UINT := [0,1,6,5];
	distanceTrack    :ARRAY[0..gvl.MAX_mover]OF LREAL;
	seqEnableTrack  :UINT;
	seqEnableUtility :UINT;
	seqDetectIdBumper:UINT;
	EnableTrack     :BOOL:=TRUE;
	EnableUtility    :BOOL := TRUE;
	DetectIdBumper  :BOOL;
	resultSettCoordmoverCommunicationCmd:BOOL;
	MoverComStatus 	:MoverCommunicationStatus;
	btnMover        :STRING;
	stMoverDetecionStatus:MoverDetectionStatus;
	Timer             :TON;
	estmatedMoverPower:POINTER TO LREAL;
	OutputForce       :POINTER TO MoverVector;
	
	i,j: INT; //Mover
	k: INT; //
	t: INT; //Track
	
	seqEnableT: INT;
	resultIniU: BOOL;
	
	bMoverEnable : ARRAY [0..gvl.MAX_MOVER] OF BOOL;
	bJoinTrackseq: BOOL;
	bMoveTrackSeq: BOOL;
	diCountSum: DINT;
	CountReset: BOOL;
	TrigSlowStop : F_TRIG;
	bPtoP_X: BOOL;
	bX600: BOOL;
	
	pSortedMovers	: ARRAY [0..GVL.MAX_MOVER] OF POINTER TO MC_PlanarMover;
	pTemp			: POINTER TO MC_PlanarMover;
	pMover_1st,pMover_2nd, pMover_3rd, pMover_4th : POINTER TO MC_PlanarMover;
	
	nJoinStep: INT;
END_VAR

VAR
	IpXpu            :I_TcIoXPlanarProcessingUnit;
	FbEnv            :FB_TcIoXPlanarEnvironment;
	Xpmover          :ARRAY [0..gvl.MAX_MOVER]OF MC_PlanarMover;
	Xpfeedback       :ARRAY [0..gvl.MAX_mover]OF U_MoverFeedback;
//	Xpfeedback       :ARRAY [0..gvl.MAX_mover]OF ARRAY [0..gvl.MAX_FEEDBACK]OF MC_Planarfeedback;
	XpTrack          :ARRAY [0..gvl.MAX_Track]OF MC_PlanarTrack;
	ConstraintXY    :ARRAY [0..gvl.MAX_mover]OF DynamicConstraint_PathXY;	
	Constratint_ZABC :ARRAY [0..gvl.MAX_mover]OF DynamicConstraint_Coordinates;
END_VAR

VAR CONSTANT
	MAX_MOVER     :UINT:=1;
	MAX_FEEDBACK  :UINT:=100;
	MAX_Track     :UINT:=7;
END_VAR

VAR CONSTANT
	INIT      :UINT:=0;
	READY     :UINT:=10;
	EXECUTE   :UINT:=1;
	BUSY      :UINT:=2;
	DONE      :UINT:=3;
	ERROR     :UINT:=4;
	ABORT     :UINT:=5;
	
	
END_VAR

VAR //StateTrackMove
	fbStateTrack : ARRAY [0..gvl.max_mover] OF FB_StateTrackMove; 
END_VAR

VAR //Keyence IO
	bSlowStop 		AT %I*	:BOOL;//Sefety PLC
	//iEipInput 		AT %I*	:ARRAY[0..50] OF INT;//EthernetIP Input
	//iEipOutput		AT %Q* 	:ARRAY[0..50] OF INT;//EthernetIP Output
	iEipInput 		AT %I*	:ARRAY[0..50] OF WORD;//EthernetIP Input
	iEipOutput		AT %Q* 	:ARRAY[0..50] OF WORD;//EthernetIP Output
	bEipInput		AT %I*	:ARRAY[0..9] OF BOOL;
	bEipOutput		AT %Q*	:ARRAY[0..9] OF BOOL;
END_VAR

update();//Mover and Track Update
callEnableT();//Track Enable
callMoveX_2m();
callEnableUtility();//fbEnv Init
//callDetectIdBumper();//Detect ID Bumper

(*
FOR i:=0 TO gvl.MAX_MOVER DO //Mover
	callEmergencyStop();
END_FOR
*)
TrigSlowStop(CLK := bSlowStop);
FOR i:=0 TO gvl.MAX_MOVER DO
	IF TrigSlowStop.Q THEN
			IF XpMover[i].MCTOPLC.STD.State = MC.MC_PLANAR_STATE.Enabled THEN
				XpMover[i].Halt(commandFeedback :=XpFeedback[i].sName.CallEmergencyStop,
					constraint := ConstraintXY[i]);
			END_IF
		RETURN;
	END_IF
END_FOR

FOR i:=0 TO gvl.MAX_MOVER DO //Mover
	callEnable();
	callReset();
	callHalt();
	calldisable();
	callMoveX();
	callMoveY();
	callMoveA();	
	callMoveB();	
	callMoveZ();
	callMoveC();	
	callJoinTrack();	
	callLeaveTrack();
	callMoveOnTrack();	

	
	fbStateTrack[i](
	Fbmover:=xpMover[i],
	fbTrack:=xptrack,
	bEmergencyStopIn:=bSlowStop);
	
END_FOR
seq_JoinTrack();

IF seqEnableUtility = done THEN
	estmatedMoverPower:= IpXpu.TcIoMover(2).ScopeAdr.GetEstimatedMoverPower();
	OutputForce:= IpXpu.TcIoMover(2).ScopeAdr.GetOutputForce();
END_IF

FOR i :=0 TO gvl.MAX_MOVER DO
	bMoverEnable[i] := (MAIN.Xpmover[i].MCTOPLC.STD.State = MC_PLANAR_STATE.Enabled);
END_FOR

IF bPtoP_X THEN
	IF bX600 THEN
		positionTargetX[0]:=600;
	ELSE
		positionTargetX[0]:=120;
	END_IF
END_IF

IF iEipInput[0].0 THEN
	iEipOutput[0].0:=TRUE;
	FOR i:=0 TO GVL.MAX_MOVER DO
	fbStateTrack[i].bMoveState:= TRUE;
	END_FOR
END_IF


IF iEipInput[0].1 THEN
	GVL.bstop:= TRUE;
ELSE
	GVL.bstop := FALSE;
END_IF

ACTION callDetectIdBumper:
(*
CASE seqDetectIdBumper OF
	
INIT:
	seqDetectIdBumper:=READY;
		
READY:
	DetectIdBumper := (seqEnableUtility = done);
	IF DetectIdBumper THEN
		IpXpu.SetStartMoverRedetection();
        seqDetectIdBumper:=11; 
	END_IF
	
11:
	stMoverDetecionStatus:= ipXpu.GetMoverDetectionStatus();
	IF stMoverDetecionStatus= MoverDetectionStatus.DetectionSuccessful THEN
		seqDetectIdBumper:=12;
	END_IF
		
12:
	Timer(IN:=TRUE , PT:=T#5S , Q=> , ET=> );
	IF timer.Q THEN
		resultSettCoordmoverCommunicationCmd:=IpXpu.SetCoordmoverCommunicationCmd(
			CoordinatedMoverCommCommand.IdentifyBTNsAndRearrangeMovers);
		seqDetectIdBumper:=13; 
	END_IF
		
13:
	MoverComStatus:=IpXpu.TcIoMover(1).GetCommunicationStatus();
	btnMover:=IpXpu.TcIoMover(1).GetIdentifiedMoverBtn();
	IF MoverComStatus= MoverCommunicationStatus.CommunicationSuccessful THEN
	   seqDetectIdBumper:= DONE;
	ELSIF MoverComStatus= MoverCommunicationStatus.CommunicationFailed THEN
	   seqDetectIdBumper:= ERROR;
	END_IF	
		
BUSY:
   (*
    IF XpFeedback[i][12].Done THEN
		seqMoveX1M[i]:=DONE;
    ELSIF Xpfeedback[i][12].Aborted THEN
		seqMoveX1M[i]:=ABORT;
	ELSIF Xpfeedback[i][12].Error THEN	
		seqMoveX1M[i]:=ERROR;
	END_IF
		//
	  *)
	  
DONE:
	IF NOT DetectIdBumper THEN
	   seqDetectIdBumper:=READY;
	END_IF
		
ERROR:
	IF NOT DetectIdBumper THEN
	   seqDetectIdBumper:=READY;
	END_IF
		
ABORT:
	IF NOT DetectIdBumper THEN
	   seqDetectIdBumper:=READY;
	END_IF
		
END_CASE

*)
END_ACTION

ACTION Calldisable:
CASE seqdisableM[i] OF

INIT:
	seqdisableM[i]:=READY;

READY:
	IF disableM [i] THEN
    	disableM [i] :=FALSE;
    	Xpmover[i].disable(commandFeedback:=XpFeedBack[i].sName.CallDisable);
	END_IF
	 
BUSY:
	IF xpFeedback[i].sName.CallDisable.Done THEN
	   disableM[i]:=FALSE;
	   seqdisableM[i]:=DONE;
	END_IF

DONE:
	IF NOT disableM[i] THEN
	   seqdisableM[i]:=READY;
	END_IF
	
END_CASE
END_ACTION

ACTION callEmergencyStop:
(*
TrigSlowStop(CLK := bSlowStop);

IF TrigSlowStop.Q THEN
	FOR i:=1 TO GVL.MAX_MOVER DO
		IF XpMover[i].MCTOPLC.STD.State = MC.MC_PLANAR_STATE.Enabled THEN
			XpMover[i].Halt(commandFeedback :=XpFeedback[i].sName.CallEmergencyStop,
				constraint := ConstraintXY[i]);
		END_IF
	END_FOR
	//RETURN;
END_IF


IF NOT bSlowStop THEN //非常停止時にHaltで停止かける
	FOR i:=1 TO GVL.MAX_MOVER DO
		IF XpMover[i].MCTOPLC.STD.State = MC.MC_PLANAR_STATE.Enabled THEN
			XpMover[i].Halt(commandFeedback :=XpFeedback[i].sName.CallEmergencyStop,
				constraint := ConstraintXY[1]);
		END_IF
	END_FOR
	
END_IF
*)
END_ACTION

ACTION CallEnable:
CASE seqEnableM[i] OF

INIT:
	seqEnableM[i]:=READY;

READY:
	IF enableM[i]THEN
		xpMover[i].Enable(commandFeedback:=XpFeedBack[i].sName.CallEnable);
		seqEnableM[i]:=BUSY;
	END_IF
		
BUSY:
	IF XpFeedback[i].sName.CallEnable.Done THEN
		seqEnableM[i]:=DONE;
    ELSIF Xpfeedback[i].sName.CallEnable.Aborted THEN
		seqEnableM[i]:=ABORT;
	ELSIF Xpfeedback[i].sName.CallEnable.Error THEN	
		seqEnableM[i]:=ERROR;
	END_IF
	
DONE:
	IF NOT enableM[i] THEN
	   seqEnableM[i]:=READY;
	END_IF
	
ERROR:
	IF NOT enableM[i] THEN
	   seqEnableM[i]:=READY;
	END_IF
	
ABORT:
	IF NOT enableM[i] THEN
	   seqenableM[i]:=READY;
	END_IF
		   	   
END_CASE
END_ACTION

ACTION callEnableT:
CASE seqEnableT OF
	INIT:
	seqEnableT:=READY;
	
	READY:
	IF EnableTrack THEN
		FOR t:=0 TO MAX_TRACK DO
			XpTrack[t].Enable(commandFeedback:=0);
		END_FOR
		seqEnableT:=DONE;
	END_IF
	DONE:
	
END_CASE
END_ACTION

ACTION callEnableUtility:
CASE seqEnableUtility OF
	
INIT:
	seqEnableUtility:=READY;	

READY:
	IF EnableUtility THEN
    	seqEnableUtility :=BUSY;
	END_IF
		
BUSY:
	resultIniU:=FbEnv.Init(bExecute:=TRUE );
	IF resultIniU THEN
		FbEnv.Init(bExecute:=FALSE );
		IpXpu:=FbEnv.TcIoXpu(nNum:= 1);
		seqEnableUtility:=DONE;
	END_IF
	
DONE:
	IF NOT EnableUtility THEN
	   seqEnableUtility:=READY;
	END_IF

ERROR:
	IF NOT EnableUtility THEN
	   seqEnableUtility:=READY;
	END_IF

ABORT:
	IF NOT EnableUtility THEN
	   seqEnableUtility:=READY;
	END_IF
		
END_CASE
END_ACTION

ACTION CallHalt:
CASE seqHaltM[i] OF

INIT:
	seqHaltM[i]:=READY;

READY:
	IF HaltM[i]THEN
		Xpmover[i].Halt(commandFeedback:=XpFeedBack[i].sName.CallHalt , 
				constraint:=0 );
		seqHaltM[i]:=BUSY;
	END_IF

BUSY:
	IF xpFeedback[i].sName.CallHalt.Done THEN
		HaltM[i]:=FALSE;
		seqHaltM[i]:=DONE;
	END_IF

DONE:
	IF NOT HaltM[i] THEN
	   seqHaltM[i]:=READY;
	END_IF
	
END_CASE
END_ACTION

ACTION callJoinTrack:
CASE seqJoinTrack[i] OF

INIT:
	seqJoinTrack[i]:=READY;	

READY:
	fbStateTrack[i].bstart:=FALSE;
	IF JoinTrack[i]THEN
		JoinTrack[i]:=FALSE;
		ConstraintXY[i].SetValuesVADJ(V:=velocity_xy[i] , A:=800 , D:=900 , J:=5000 );
	 	Xpmover[i].JoinTrack(commandFeedback:=xpFeedback[i].sName.CallJoinTrack , 
                          targetTrack:= XpTrack[numbertrack[i]],
                           constraint:= ConstraintXY[i],
                           options:=0 );
		seqJoinTrack[i]:=BUSY;
	END_IF	
		
BUSY:
	IF XpFeedback[i].sName.CallJoinTrack.Done THEN
		seqJoinTrack[i]:=DONE;
    ELSIF Xpfeedback[i].sName.CallJoinTrack.Aborted THEN
		seqJoinTrack[i]:=ABORT;
	ELSIF Xpfeedback[i].sName.CallJoinTrack.Error THEN	
		seqJoinTrack[i]:=ERROR;
	END_IF
	
DONE:
	IF NOT JoinTrack[i] THEN
		fbStateTrack[i].bstart:=TRUE;
		gvl.bBusyA:=FALSE;
		gvl.bBusyB:=FALSE;
		gvl.bDoneA:=FALSE;
		gvl.bDoneB:=FALSE;
	   seqJoinTrack[i]:=READY;
	END_IF

ERROR:
	IF NOT JoinTrack[i] THEN
	   seqJoinTrack[i]:=READY;
	END_IF

ABORT:
	IF NOT JoinTrack[i] THEN
	   seqJoinTrack[i]:=READY;
	END_IF
		
END_CASE
END_ACTION

ACTION callLeaveTrack:
CASE seqLeaveTrack[i] OF

INIT:
	seqLeaveTrack[i]:=READY;	

READY:
	IF LeaveTrack[i]THEN
		ConstraintXY[i].SetValuesVADJ(
			V:=velocity_xy[i],
			A:=20000,
			D:=20000,
			J:=200000 );
		PositionXYC[i].SetValuesXYC(
			x:=PositionTargetX[i], 
            y:=PositionTargetY[i], 
            c:=PositionTargetC[i]);
		Xpmover[i].LeaveTrack(
			commandFeedback:=xpFeedback[i].sName.CallLeaveTrack,
				targetPosition:=PositionXYC[i] , 
				constraint:= ConstraintXY[i],
				options:=0 );
		seqLeaveTrack[i]:=BUSY;
	END_IF
		
BUSY:
    IF XpFeedback[i].sName.CallLeaveTrack.Done THEN
		seqLeaveTrack[i]:=DONE;
    ELSIF Xpfeedback[i].sName.CallLeaveTrack.Aborted THEN
		seqLeaveTrack[i]:=ABORT;
	ELSIF Xpfeedback[i].sName.CallLeaveTrack.Error THEN	
		seqLeaveTrack[i]:=ERROR;
	END_IF
	
DONE:
	IF NOT LeaveTrack[i] THEN
	   seqLeaveTrack[i]:=READY;
	END_IF
	
ERROR:
	IF NOT LeaveTrack[i] THEN
	   seqLeaveTrack[i]:=READY;
	END_IF
	
ABORT:
	IF NOT LeaveTrack[i] THEN
	   seqLeaveTrack[i]:=READY;
	END_IF
		
END_CASE
END_ACTION

ACTION callMoveA:
CASE seqMoveAM[i] OF
	
INIT:
	seqMoveAM[i]:=READY;
	Constratint_ZABC[i].SetLimit(
		Coordinate:= Coord_Mcs_A1, 
		V:= 100 , 
		A:= 100 , 
		D:= 100, 
		J:= 1000);
	
READY:
	IF moveAM[i]THEN
		MoveAM[i] := FALSE;
		Constratint_ZABC[i].AddLimit(
			Coordinate:= Coord_Mcs_A1, 
			V:= 100 , 
			A:= 100 , 
			D:= 100, 
			J:= 1000);
		Xpmover[i].MoveA(
			commandFeedback:=xpFeedback[i].sName.CallMoveA , 
			targetPosition:=positionTargetA[i] , 
			constraint:=ConstraTINT_zabc[i]);
		seqMoveAM[i]:=BUSY;
	END_IF
		
BUSY:
    IF XpFeedback[i].sName.CallMoveA.Done THEN
		seqMoveAM[i]:=DONE;
    ELSIF Xpfeedback[i].sName.CallMoveA.Aborted THEN
		seqMoveAM[i]:=ABORT;
	ELSIF Xpfeedback[i].sName.CallMoveA.Error THEN	
		seqMoveAM[i]:=ERROR;
	END_IF
	
DONE:
	IF NOT MoveAM[i] THEN
	   seqMoveAM[i]:=READY;
	END_IF
		
ERROR:
	IF NOT MoveAM[i] THEN
	   seqMoveAM[i]:=READY;
	END_IF

ABORT:
	IF NOT MoveAM[i] THEN
	   seqMoveAM[i]:=READY;
	END_IF
		
END_CASE
END_ACTION

ACTION callMoveB:
CASE seqMoveBM[i] OF
	
INIT:
	seqMoveBM[i]:=READY;
	Constratint_ZABC[i].SetLimit(
		Coordinate:= Coord_Mcs_B1, 
		V:= 100 , 
		A:= 100 , 
		D:= 100, 
		J:= 1000);
	
 READY:
	IF moveBM[i]THEN
		MoveBM[i] := FALSE;
		Constratint_ZABC[i].AddLimit(
			Coordinate:= Coord_Mcs_B1, 
			V:= 100 , 
			A:= 100 , 
			D:= 100, 
			J:= 1000);
		Xpmover[i].MoveB(
			commandFeedback:=xpFeedback[i].sName.CallMoveB , 
			targetPosition:=positionTargetB[i] , 
			constraint:=ConstraTINT_zabc[i]);
		seqMoveBM[i]:=BUSY;
	END_IF

BUSY:
	IF XpFeedback[i].sName.CallMoveA.Done THEN
		seqMoveBM[i]:=DONE;
	ELSIF Xpfeedback[i].sName.CallMoveB.Aborted THEN
		seqMoveBM[i]:=ABORT;
	ELSIF Xpfeedback[i].sName.CallMoveB.Error THEN	
		seqMoveBM[i]:=ERROR;
	END_IF
	
DONE:
	IF NOT MoveBM[i] THEN
	   seqMoveBM[i]:=READY;	   
	END_IF
	
ERROR:
	IF NOT MoveBM[i] THEN
	   seqMoveBM[i]:=READY;
	END_IF
	
ABORT:
	IF NOT MoveBM[i] THEN
	   seqMoveBM[i]:=READY;
	END_IF
		
END_CASE
END_ACTION

ACTION callMoveC:
CASE seqMoveCM[i] OF
	
